KUKA KRL program: EPS_2_25862_MH04_A_20251016040658.src

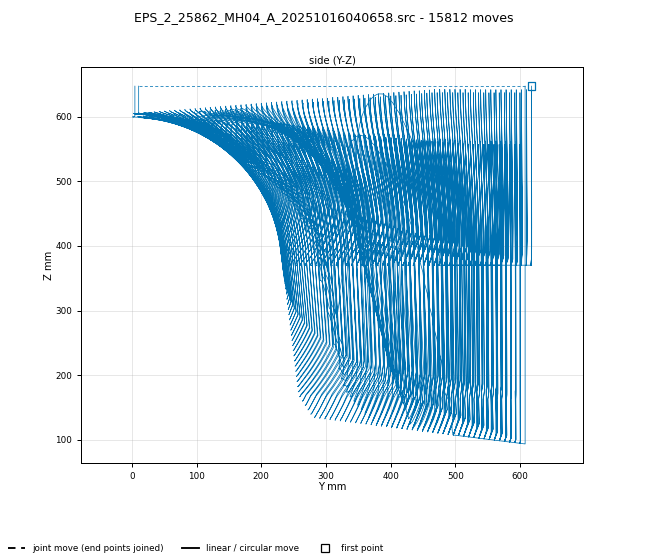
[picture p0: tool path of EPS_2_25862_MH04_A_20251016040658.src, 15812 of 15814 moves have a stored position in this frame; points joined in program order, loops and branches not executed]
&ACCESS RVP
&REL 4
&COMMENT QRS 19112012
&PARAM EDITMASK = *
DEF PART()
EXT BAS (BAS_COMMAND :IN,REAL :IN )
INT I
BAS (#INITMOV,0 )

;KUKA QRS Post kuka4.cps  Date:22-06-2017 !

File_ID=2885

QRS_PRE_INIT()

;Init var - Until changes are made in qrs_pre_init
Outlet_Square_prg=0
Inlet_1_Square_prg=0
Inlet_2_Square_prg=0
Inlet_3_Square_prg=0
Inlet_4_Square_prg=0
Inlet_5_Square_prg=0

Outlet_1={X 0.000, Y 466.000, Z 408.500, B 0.000, E1 0.000 }
Inlet_1={X 0.000, Y 522.780, Z 374.000, B 0.000, E1 180.000 }
Inlet_2={X 0.000, Y 522.780, Z 374.000, B 0.000, E1 270.000 }
Outlet_1_type=457
Inlet_1_type=366
Inlet_2_type=366
;QRS#1=Sidecore dimensions
;QRS#2=450-18" Concrete
;QRS#3=375-15" PVC SDR 35
;QRS#4=375-15" PVC SDR 35
;QRS#5=
;QRS#6=
;QRS#7=
;QRS#8=
;QRS#9=28A PSX-2
;QRS#10=20Y PSX
;QRS#11=20Y PSX
;QRS#12=
;QRS#13=
;QRS#14=
;QRS#15=
;QRS#16=1220x127x991 3,25'
;QRS#17=EPS Height
;QRS#18=637
;QRS#19=*
;QRS#20= UPDATED VERSION 22-06-2017
;QRS#21=*
Outlet_Square=0250
Inlet_1_Square=0250
Inlet_2_Square=0250
Inlet_3_Square=0
Inlet_4_Square=0
Inlet_5_Square=0
Mill_Square=1
Outlet_Square_Prg=274
Inlet_1_Square_prg=252
Inlet_2_Square_prg=252

QRS_INIT()

$ADVANCE=5

; T1
PTP {E1 171.055,E2 171.055}
PTP {X 0,Y 617.763,A -85,B 0,C 180,E1 171.055,E2 171.055,E3 0,E4 0,E5 0,E6 0}
QRS_SPEED_INIT()
LIN {X 0,Y 617.763,Z 647,A -85,B 0,C 180,E1 171.055,E2 171.055,E3 0,E4 0,E5 0,E6 0} C_VEL
LIN {X 0,Y 617.763,Z 372.16,A -85,B 0,C 180,E1 171.055,E2 171.055} C_VEL
LIN {X 0,Y 617.801,Z 370.16,A -85,B 0,C 180,E1 171.241,E2 171.241} C_VEL
LIN {X 0,Y 617.985,Z 370.16,A -85,B 0,C 180,E1 171.886,E2 171.886} C_VEL
LIN {X 0,Y 618.056,Z 370.16,A -85,B 0,C 180,E1 176.532,E2 176.532} C_VEL
LIN {X 0,Y 618.006,Z 370.16,A -85,B 0,C 180,E1 181.155,E2 181.155} C_VEL
LIN {X 0,Y 617.998,Z 370.16,A -85,B 0,C 180,E1 185.786,E2 185.786} C_VEL
LIN {X 0,Y 617.999,Z 370.16,A -85,B 0,C 180,E1 190.456,E2 190.456} C_VEL
LIN {X 0,Y 617.933,Z 370.16,A -85,B 0,C 180,E1 195.198,E2 195.198} C_VEL
LIN {X 0,Y 617.958,Z 370.16,A -85,B 0,C 180,E1 200.048,E2 200.048} C_VEL
LIN {X 0,Y 617.454,Z 370.16,A -85,B 0,C 180,E1 202.548,E2 202.548} C_VEL
LIN {X 0,Y 617.878,Z 370.16,A -85,B 0,C 180,E1 205.058,E2 205.058} C_VEL
LIN {X 0,Y 617.387,Z 370.16,A -85,B 0,C 180,E1 207.661,E2 207.661} C_VEL
LIN {X 0,Y 617.859,Z 370.16,A -85,B 0,C 180,E1 210.279,E2 210.279} C_VEL
LIN {X 0,Y 617.331,Z 370.16,A -85,B 0,C 180,E1 213.026,E2 213.026} C_VEL
LIN {X 0,Y 617.826,Z 370.16,A -85,B 0,C 180,E1 215.797,E2 215.797} C_VEL
LIN {X 0,Y 617.905,Z 370.16,A -85,B 0,C 180,E1 218.696,E2 218.696} C_VEL
LIN {X 0,Y 617.423,Z 370.16,A -85,B 0,C 180,E1 221.762,E2 221.762} C_VEL
LIN {X 0,Y 617.856,Z 370.16,A -85,B 0,C 180,E1 224.903,E2 224.903} C_VEL
LIN {X 0,Y 617.741,Z 370.16,A -85,B 0,C 180,E1 228.278,E2 228.278} C_VEL
LIN {X 0,Y 617.537,Z 370.16,A -85,B 0,C 180,E1 231.278,E2 231.278} C_VEL
LIN {X 0,Y 617.566,Z 370.16,A -85,B 0,C 180,E1 231.901,E2 231.901} C_VEL
LIN {X 0,Y 617.813,Z 370.16,A -85,B 0,C 180,E1 234.203,E2 234.203} C_VEL
LIN {X 0,Y 617.312,Z 370.16,A -85,B 0,C 180,E1 236.974,E2 236.974} C_VEL
LIN {X 0,Y 617.839,Z 370.16,A -85,B 0,C 180,E1 239.721,E2 239.721} C_VEL
LIN {X 0,Y 618.074,Z 370.16,A -85,B 0,C 180,E1 244.633,E2 244.633} C_VEL
LIN {X 0,Y 617.706,Z 370.16,A -85,B 0,C 180,E1 244.776,E2 244.776} C_VEL
LIN {X 0,Y 617.081,Z 370.236,A -85,B 0,C 180,E1 244.869,E2 244.869} C_VEL
LIN {X 0,Y 617.72,Z 382.151,A -85,B 0,C 180,E1 245.046,E2 245.046} C_VEL
LIN {X 0,Y 617.911,Z 419.432,A -85,B 0,C 180,E1 245.531,E2 245.531} C_VEL
LIN {X 0,Y 617.851,Z 429.801,A -85,B 0,C 180,E1 245.698,E2 245.698} C_VEL
LIN {X 0,Y 617.803,Z 439.075,A -85,B 0,C 180,E1 245.882,E2 245.882} C_VEL
LIN {X 0,Y 617.897,Z 451.685,A -85,B 0,C 180,E1 246.204,E2 246.204} C_VEL
LIN {X 0,Y 617.827,Z 462.897,A -85,B 0,C 180,E1 246.539,E2 246.539} C_VEL
LIN {X 0,Y 617.935,Z 474.971,A -85,B 0,C 180,E1 246.971,E2 246.971} C_VEL
LIN {X 0,Y 617.943,Z 485.368,A -85,B 0,C 180,E1 247.392,E2 247.392} C_VEL
LIN {X 0,Y 617.874,Z 495.678,A -85,B 0,C 180,E1 247.859,E2 247.859} C_VEL
LIN {X 0,Y 617.945,Z 506.347,A -85,B 0,C 180,E1 248.407,E2 248.407} C_VEL
LIN {X 0,Y 617.966,Z 517.222,A -85,B 0,C 180,E1 249.028,E2 249.028} C_VEL
LIN {X 0,Y 617.937,Z 527.03,A -85,B 0,C 180,E1 249.644,E2 249.644} C_VEL
LIN {X 0,Y 617.951,Z 536.534,A -85,B 0,C 180,E1 250.302,E2 250.302} C_VEL
LIN {X 0,Y 617.957,Z 545.725,A -85,B 0,C 180,E1 250.999,E2 250.999} C_VEL
LIN {X 0,Y 617.962,Z 554.652,A -85,B 0,C 180,E1 251.74,E2 251.74} C_VEL
LIN {X 0,Y 617.941,Z 563.035,A -85,B 0,C 180,E1 252.497,E2 252.497} C_VEL
LIN {X 0,Y 617.895,Z 570.428,A -85,B 0,C 180,E1 253.221,E2 253.221} C_VEL
LIN {X 0,Y 617.949,Z 578.128,A -85,B 0,C 180,E1 254.047,E2 254.047} C_VEL
LIN {X 0,Y 617.971,Z 584.666,A -85,B 0,C 180,E1 254.803,E2 254.803} C_VEL
LIN {X 0,Y 617.883,Z 591.779,A -85,B 0,C 180,E1 255.697,E2 255.697} C_VEL
LIN {X 0,Y 617.867,Z 598.243,A -85,B 0,C 180,E1 256.59,E2 256.59} C_VEL
LIN {X 0,Y 617.969,Z 604.103,A -85,B 0,C 180,E1 257.481,E2 257.481} C_VEL
LIN {X 0,Y 617.879,Z 609.465,A -85,B 0,C 180,E1 258.365,E2 258.365} C_VEL
LIN {X 0,Y 617.831,Z 615.768,A -85,B 0,C 180,E1 259.542,E2 259.542} C_VEL
LIN {X 0,Y 617.911,Z 619.334,A -85,B 0,C 180,E1 260.281,E2 260.281} C_VEL
LIN {X 0,Y 617.927,Z 624.37,A -85,B 0,C 180,E1 261.452,E2 261.452} C_VEL
LIN {X 0,Y 617.83,Z 627.758,A -85,B 0,C 180,E1 262.351,E2 262.351} C_VEL
LIN {X 0,Y 617.871,Z 630.79,A -85,B 0,C 180,E1 263.283,E2 263.283} C_VEL
LIN {X 0,Y 617.981,Z 633.385,A -85,B 0,C 180,E1 264.214,E2 264.214} C_VEL
LIN {X 0,Y 617.916,Z 634.618,A -85,B 0,C 180,E1 264.678,E2 264.678} C_VEL
LIN {X 0,Y 617.792,Z 636.669,A -85,B 0,C 180,E1 265.605,E2 265.605} C_VEL
LIN {X 0,Y 617.811,Z 638.259,A -85,B 0,C 180,E1 266.531,E2 266.531} C_VEL
LIN {X 0,Y 617.948,Z 639.966,A -85,B 0,C 180,E1 267.92,E2 267.92} C_VEL
LIN {X 0,Y 617.798,Z 640.661,A -85,B 0,C 180,E1 268.845,E2 268.845} C_VEL
LIN {X 0,Y 617.834,Z 640.908,A -85,B 0,C 180,E1 270.232,E2 270.232} C_VEL
LIN {X 0,Y 617.983,Z 640.61,A -85,B 0,C 180,E1 271.156,E2 271.156} C_VEL
LIN {X 0,Y 617.815,Z 639.475,A -85,B 0,C 180,E1 272.544,E2 272.544} C_VEL
LIN {X 0,Y 617.845,Z 638.248,A -85,B 0,C 180,E1 273.469,E2 273.469} C_VEL
LIN {X 0,Y 617.914,Z 637.45,A -85,B 0,C 180,E1 273.932,E2 273.932} C_VEL
LIN {X 0,Y 617.842,Z 634.634,A -85,B 0,C 180,E1 275.324,E2 275.324} C_VEL
LIN {X 0,Y 617.779,Z 632.188,A -85,B 0,C 180,E1 276.254,E2 276.254} C_VEL
LIN {X 0,Y 617.944,Z 627.726,A -85,B 0,C 180,E1 277.649,E2 277.649} C_VEL
LIN {X 0,Y 617.874,Z 623.347,A -85,B 0,C 180,E1 278.796,E2 278.796} C_VEL
LIN {X 0,Y 617.822,Z 619.616,A -85,B 0,C 180,E1 279.666,E2 279.666} C_VEL
LIN {X 0,Y 617.937,Z 614.253,A -85,B 0,C 180,E1 280.751,E2 280.751} C_VEL
LIN {X 0,Y 617.944,Z 609.445,A -85,B 0,C 180,E1 281.634,E2 281.634} C_VEL
LIN {X 0,Y 617.865,Z 602.193,A -85,B 0,C 180,E1 282.818,E2 282.818} C_VEL
LIN {X 0,Y 617.94,Z 596.131,A -85,B 0,C 180,E1 283.707,E2 283.707} C_VEL
LIN {X 0,Y 617.957,Z 589.464,A -85,B 0,C 180,E1 284.6,E2 284.6} C_VEL
LIN {X 0,Y 617.88,Z 581.509,A -85,B 0,C 180,E1 285.571,E2 285.571} C_VEL
LIN {X 0,Y 617.913,Z 574.458,A -85,B 0,C 180,E1 286.356,E2 286.356} C_VEL
LIN {X 0,Y 617.964,Z 566.289,A -85,B 0,C 180,E1 287.188,E2 287.188} C_VEL
LIN {X 0,Y 617.928,Z 559.146,A -85,B 0,C 180,E1 287.864,E2 287.864} C_VEL
LIN {X 0,Y 617.92,Z 550.267,A -85,B 0,C 180,E1 288.633,E2 288.633} C_VEL
LIN {X 0,Y 617.942,Z 541.357,A -85,B 0,C 180,E1 289.339,E2 289.339} C_VEL
LIN {X 0,Y 617.96,Z 532.851,A -85,B 0,C 180,E1 289.96,E2 289.96} C_VEL
LIN {X 0,Y 617.949,Z 523.456,A -85,B 0,C 180,E1 290.588,E2 290.588} C_VEL
LIN {X 0,Y 617.919,Z 513.262,A -85,B 0,C 180,E1 291.207,E2 291.207} C_VEL
LIN {X 0,Y 617.945,Z 503.396,A -85,B 0,C 180,E1 291.75,E2 291.75} C_VEL
LIN {X 0,Y 617.963,Z 492.338,A -85,B 0,C 180,E1 292.294,E2 292.294} C_VEL
LIN {X 0,Y 617.929,Z 481.553,A -85,B 0,C 180,E1 292.769,E2 292.769} C_VEL
LIN {X 0,Y 617.813,Z 471.413,A -85,B 0,C 180,E1 293.169,E2 293.169} C_VEL
LIN {X 0,Y 617.936,Z 458.266,A -85,B 0,C 180,E1 293.602,E2 293.602} C_VEL
LIN {X 0,Y 617.915,Z 446.913,A -85,B 0,C 180,E1 293.922,E2 293.922} C_VEL
LIN {X 0,Y 617.746,Z 436.06,A -85,B 0,C 180,E1 294.184,E2 294.184} C_VEL
LIN {X 0,Y 617.908,Z 424.188,A -85,B 0,C 180,E1 294.398,E2 294.398} C_VEL
LIN {X 0,Y 617.873,Z 406.799,A -85,B 0,C 180,E1 294.638,E2 294.638} C_VEL
LIN {X 0,Y 617.621,Z 379.189,A -85,B 0,C 180,E1 294.995,E2 294.995} C_VEL
LIN {X 0,Y 617.066,Z 370.16,A -85,B 0,C 180,E1 295.133,E2 295.133} C_VEL
LIN {X 0,Y 617.707,Z 370.16,A -85,B 0,C 180,E1 295.225,E2 295.225} C_VEL
LIN {X 0,Y 618.075,Z 370.16,A -85,B 0,C 180,E1 295.369,E2 295.369} C_VEL
LIN {X 0,Y 617.989,Z 370.16,A -85,B 0,C 180,E1 297.632,E2 297.632} C_VEL
LIN {X 0,Y 617.43,Z 370.16,A -85,B 0,C 180,E1 300.303,E2 300.303} C_VEL
LIN {X 0,Y 617.934,Z 370.16,A -85,B 0,C 180,E1 302.99,E2 302.99} C_VEL
LIN {X 0,Y 617.673,Z 370.16,A -85,B 0,C 180,E1 305.808,E2 305.808} C_VEL
LIN {X 0,Y 617.667,Z 370.16,A -85,B 0,C 180,E1 308.111,E2 308.111} C_VEL
LIN {X 0,Y 617.76,Z 370.16,A -85,B 0,C 180,E1 311.734,E2 311.734} C_VEL
LIN {X 0,Y 617.402,Z 370.16,A -85,B 0,C 180,E1 315.055,E2 315.055} C_VEL
LIN {X 0,Y 617.766,Z 370.16,A -85,B 0,C 180,E1 318.276,E2 318.276} C_VEL
LIN {X 0,Y 617.372,Z 370.16,A -85,B 0,C 180,E1 321.925,E2 321.925} C_VEL
LIN {X 0,Y 617.835,Z 370.16,A -85,B 0,C 180,E1 324.203,E2 324.203} C_VEL
LIN {X 0,Y 617.363,Z 370.16,A -85,B 0,C 180,E1 326.976,E2 326.976} C_VEL
LIN {X 0,Y 617.895,Z 370.16,A -85,B 0,C 180,E1 329.723,E2 329.723} C_VEL
LIN {X 0,Y 617.432,Z 370.16,A -85,B 0,C 180,E1 332.342,E2 332.342} C_VEL
LIN {X 0,Y 617.927,Z 370.16,A -85,B 0,C 180,E1 334.945,E2 334.945} C_VEL
LIN {X 0,Y 618.05,Z 370.16,A -85,B 0,C 180,E1 339.647,E2 339.647} C_VEL
LIN {X 0,Y 617.925,Z 370.16,A -85,B 0,C 180,E1 339.797,E2 339.797} C_VEL
LIN {X 0,Y 617.569,Z 370.202,A -85,B 0,C 180,E1 339.878,E2 339.878} C_VEL
LIN {X 0,Y 617.849,Z 384.179,A -85,B 0,C 180,E1 340.078,E2 340.078} C_VEL
LIN {X 0,Y 617.994,Z 396.248,A -85,B 0,C 180,E1 340.32,E2 340.32} C_VEL
LIN {X 0,Y 618.025,Z 406.56,A -85,B 0,C 180,E1 340.58,E2 340.58} C_VEL
LIN {X 0,Y 617.971,Z 415.883,A -85,B 0,C 180,E1 340.858,E2 340.858} C_VEL
LIN {X 0,Y 617.923,Z 423.433,A -85,B 0,C 180,E1 341.114,E2 341.114} C_VEL
LIN {X 0,Y 617.995,Z 433.283,A -85,B 0,C 180,E1 341.505,E2 341.505} C_VEL
LIN {X 0,Y 617.986,Z 442.714,A -85,B 0,C 180,E1 341.929,E2 341.929} C_VEL
LIN {X 0,Y 617.95,Z 450.65,A -85,B 0,C 180,E1 342.327,E2 342.327} C_VEL
LIN {X 0,Y 617.997,Z 459.127,A -85,B 0,C 180,E1 342.801,E2 342.801} C_VEL
LIN {X 0,Y 617.99,Z 467.334,A -85,B 0,C 180,E1 343.309,E2 343.309} C_VEL
LIN {X 0,Y 617.994,Z 476.018,A -85,B 0,C 180,E1 343.905,E2 343.905} C_VEL
LIN {X 0,Y 617.979,Z 483.981,A -85,B 0,C 180,E1 344.508,E2 344.508} C_VEL
LIN {X 0,Y 617.963,Z 491.14,A -85,B 0,C 180,E1 345.102,E2 345.102} C_VEL
LIN {X 0,Y 617.968,Z 497.738,A -85,B 0,C 180,E1 345.699,E2 345.699} C_VEL
LIN {X 0,Y 618.003,Z 505.227,A -85,B 0,C 180,E1 346.443,E2 346.443} C_VEL
LIN {X 0,Y 617.949,Z 512.018,A -85,B 0,C 180,E1 347.184,E2 347.184} C_VEL
LIN {X 0,Y 617.926,Z 519.37,A -85,B 0,C 180,E1 348.071,E2 348.071} C_VEL
LIN {X 0,Y 617.997,Z 525.839,A -85,B 0,C 180,E1 348.956,E2 348.956} C_VEL
LIN {X 0,Y 617.946,Z 531.027,A -85,B 0,C 180,E1 349.739,E2 349.739} C_VEL
LIN {X 0,Y 617.876,Z 535.713,A -85,B 0,C 180,E1 350.519,E2 350.519} C_VEL
LIN {X 0,Y 617.912,Z 539.315,A -85,B 0,C 180,E1 351.182,E2 351.182} C_VEL
LIN {X 0,Y 617.988,Z 543.836,A -85,B 0,C 180,E1 352.119,E2 352.119} C_VEL
LIN {X 0,Y 617.903,Z 546.855,A -85,B 0,C 180,E1 352.817,E2 352.817} C_VEL
LIN {X 0,Y 617.832,Z 550.397,A -85,B 0,C 180,E1 353.747,E2 353.747} C_VEL
LIN {X 0,Y 617.917,Z 553.348,A -85,B 0,C 180,E1 354.677,E2 354.677} C_VEL
LIN {X 0,Y 617.967,Z 555.788,A -85,B 0,C 180,E1 355.605,E2 355.605} C_VEL
LIN {X 0,Y 617.847,Z 557.776,A -85,B 0,C 180,E1 356.531,E2 356.531} C_VEL
LIN {X 0,Y 617.856,Z 559.249,A -85,B 0,C 180,E1 357.457,E2 357.457} C_VEL
LIN {X 0,Y 617.914,Z 559.779,A -85,B 0,C 180,E1 357.92,E2 357.92} C_VEL
LIN {X 0,Y 617.944,Z 560.559,A -85,B 0,C 180,E1 358.845,E2 358.845} C_VEL
LIN {X 0,Y 617.88,Z 560.798,A -85,B 0,C 180,E1 359.307,E2 359.307} C_VEL
LIN {X 0,Y 617.825,Z 560.9,A -85,B 0,C 180,E1 360.231,E2 360.231} C_VEL
LIN {X 0,Y 617.894,Z 560.509,A -85,B 0,C 180,E1 361.156,E2 361.156} C_VEL
LIN {X 0,Y 617.881,Z 559.137,A -85,B 0,C 180,E1 362.543,E2 362.543} C_VEL
LIN {X 0,Y 617.822,Z 557.63,A -85,B 0,C 180,E1 363.469,E2 363.469} C_VEL
LIN {X 0,Y 617.899,Z 555.598,A -85,B 0,C 180,E1 364.395,E2 364.395} C_VEL
LIN {X 0,Y 617.955,Z 553.067,A -85,B 0,C 180,E1 365.322,E2 365.322} C_VEL
LIN {X 0,Y 617.87,Z 550.053,A -85,B 0,C 180,E1 366.252,E2 366.252} C_VEL
LIN {X 0,Y 617.941,Z 545.458,A -85,B 0,C 180,E1 367.415,E2 367.415} C_VEL
LIN {X 0,Y 617.978,Z 542.3,A -85,B 0,C 180,E1 368.115,E2 368.115} C_VEL
LIN {X 0,Y 617.885,Z 537.344,A -85,B 0,C 180,E1 369.091,E2 369.091} C_VEL
LIN {X 0,Y 617.884,Z 534.05,A -85,B 0,C 180,E1 369.676,E2 369.676} C_VEL
LIN {X 0,Y 617.956,Z 529.189,A -85,B 0,C 180,E1 370.457,E2 370.457} C_VEL
LIN {X 0,Y 617.992,Z 524.162,A -85,B 0,C 180,E1 371.191,E2 371.191} C_VEL
LIN {X 0,Y 617.927,Z 518.64,A -85,B 0,C 180,E1 371.929,E2 371.929} C_VEL
LIN {X 0,Y 617.936,Z 512.535,A -85,B 0,C 180,E1 372.668,E2 372.668} C_VEL
LIN {X 0,Y 617.996,Z 505.794,A -85,B 0,C 180,E1 373.408,E2 373.408} C_VEL
LIN {X 0,Y 617.987,Z 499.923,A -85,B 0,C 180,E1 374.003,E2 374.003} C_VEL
LIN {X 0,Y 617.964,Z 493.532,A -85,B 0,C 180,E1 374.6,E2 374.6} C_VEL
LIN {X 0,Y 617.969,Z 486.545,A -85,B 0,C 180,E1 375.197,E2 375.197} C_VEL
LIN {X 0,Y 617.969,Z 478.994,A -85,B 0,C 180,E1 375.788,E2 375.788} C_VEL
LIN {X 0,Y 618.002,Z 470.17,A -85,B 0,C 180,E1 376.412,E2 376.412} C_VEL
LIN {X 0,Y 617.987,Z 463.836,A -85,B 0,C 180,E1 376.824,E2 376.824} C_VEL
LIN {X 0,Y 617.993,Z 454.31,A -85,B 0,C 180,E1 377.382,E2 377.382} C_VEL
LIN {X 0,Y 617.954,Z 446.299,A -85,B 0,C 180,E1 377.806,E2 377.806} C_VEL
LIN {X 0,Y 618.005,Z 437.901,A -85,B 0,C 180,E1 378.203,E2 378.203} C_VEL
LIN {X 0,Y 617.997,Z 428.224,A -85,B 0,C 180,E1 378.609,E2 378.609} C_VEL
LIN {X 0,Y 617.916,Z 419.62,A -85,B 0,C 180,E1 378.929,E2 378.929} C_VEL
LIN {X 0,Y 617.991,Z 410.198,A -85,B 0,C 180,E1 379.228,E2 379.228} C_VEL
LIN {X 0,Y 617.991,Z 400.635,A -85,B 0,C 180,E1 379.486,E2 379.486} C_VEL
LIN {X 0,Y 617.933,Z 390.91,A -85,B 0,C 180,E1 379.704,E2 379.704} C_VEL
LIN {X 0,Y 617.689,Z 380.946,A -85,B 0,C 180,E1 379.884,E2 379.884} C_VEL
LIN {X 0,Y 617.047,Z 370.16,A -85,B 0,C 180,E1 380.058,E2 380.058} C_VEL
LIN {X 0,Y 618.002,Z 370.16,A -85,B 0,C 180,E1 380.355,E2 380.355} C_VEL
LIN {X 0,Y 617.929,Z 370.16,A -85,B 0,C 180,E1 385.055,E2 385.055} C_VEL
LIN {X 0,Y 617.437,Z 370.16,A -85,B 0,C 180,E1 387.658,E2 387.658} C_VEL
LIN {X 0,Y 617.899,Z 370.16,A -85,B 0,C 180,E1 390.277,E2 390.277} C_VEL
LIN {X 0,Y 617.367,Z 370.16,A -85,B 0,C 180,E1 393.024,E2 393.024} C_VEL
LIN {X 0,Y 617.838,Z 370.16,A -85,B 0,C 180,E1 395.797,E2 395.797} C_VEL
LIN {X 0,Y 617.935,Z 370.16,A -85,B 0,C 180,E1 398.693,E2 398.693} C_VEL
LIN {X 0,Y 617.441,Z 370.16,A -85,B 0,C 180,E1 401.76,E2 401.76} C_VEL
LIN {X 0,Y 617.851,Z 370.16,A -85,B 0,C 180,E1 404.903,E2 404.903} C_VEL
LIN {X 0,Y 617.765,Z 370.16,A -85,B 0,C 180,E1 408.275,E2 408.275} C_VEL
LIN {X 0,Y 617.553,Z 370.16,A -85,B 0,C 180,E1 411.278,E2 411.278} C_VEL
LIN {X 0,Y 617.579,Z 370.16,A -85,B 0,C 180,E1 411.9,E2 411.9} C_VEL
LIN {X 0,Y 617.823,Z 370.16,A -85,B 0,C 180,E1 414.202,E2 414.202} C_VEL
LIN {X 0,Y 617.352,Z 370.16,A -85,B 0,C 180,E1 416.975,E2 416.975} C_VEL
LIN {X 0,Y 617.884,Z 370.16,A -85,B 0,C 180,E1 419.722,E2 419.722} C_VEL
LIN {X 0,Y 617.423,Z 370.16,A -85,B 0,C 180,E1 422.341,E2 422.341} C_VEL
LIN {X 0,Y 617.919,Z 370.16,A -85,B 0,C 180,E1 424.944,E2 424.944} C_VEL
LIN {X 0,Y 618.043,Z 370.16,A -85,B 0,C 180,E1 429.646,E2 429.646} C_VEL
LIN {X 0,Y 617.917,Z 370.16,A -85,B 0,C 180,E1 429.796,E2 429.796} C_VEL
LIN {X 0,Y 617.553,Z 370.168,A -85,B 0,C 180,E1 429.877,E2 429.877} C_VEL
LIN {X 0,Y 617.839,Z 384.153,A -85,B 0,C 180,E1 430.077,E2 430.077} C_VEL
LIN {X 0,Y 617.985,Z 395.303,A -85,B 0,C 180,E1 430.298,E2 430.298} C_VEL
LIN {X 0,Y 618.023,Z 406.525,A -85,B 0,C 180,E1 430.579,E2 430.579} C_VEL
LIN {X 0,Y 617.975,Z 415.849,A -85,B 0,C 180,E1 430.857,E2 430.857} C_VEL
LIN {X 0,Y 617.927,Z 423.396,A -85,B 0,C 180,E1 431.113,E2 431.113} C_VEL
LIN {X 0,Y 618.007,Z 433.84,A -85,B 0,C 180,E1 431.53,E2 431.53} C_VEL
LIN {X 0,Y 617.989,Z 442.695,A -85,B 0,C 180,E1 431.929,E2 431.929} C_VEL
LIN {X 0,Y 617.954,Z 450.641,A -85,B 0,C 180,E1 432.326,E2 432.326} C_VEL
LIN {X 0,Y 618,Z 459.118,A -85,B 0,C 180,E1 432.801,E2 432.801} C_VEL
LIN {X 0,Y 617.992,Z 467.324,A -85,B 0,C 180,E1 433.308,E2 433.308} C_VEL
LIN {X 0,Y 617.996,Z 476.144,A -85,B 0,C 180,E1 433.914,E2 433.914} C_VEL
LIN {X 0,Y 617.979,Z 483.974,A -85,B 0,C 180,E1 434.507,E2 434.507} C_VEL
LIN {X 0,Y 617.962,Z 491.135,A -85,B 0,C 180,E1 435.101,E2 435.101} C_VEL
LIN {X 0,Y 617.967,Z 497.734,A -85,B 0,C 180,E1 435.698,E2 435.698} C_VEL
LIN {X 0,Y 618.001,Z 505.223,A -85,B 0,C 180,E1 436.443,E2 436.443} C_VEL
LIN {X 0,Y 617.948,Z 512.014,A -85,B 0,C 180,E1 437.183,E2 437.183} C_VEL
LIN {X 0,Y 617.925,Z 519.367,A -85,B 0,C 180,E1 438.07,E2 438.07} C_VEL
LIN {X 0,Y 617.996,Z 525.836,A -85,B 0,C 180,E1 438.956,E2 438.956} C_VEL
LIN {X 0,Y 617.946,Z 531.023,A -85,B 0,C 180,E1 439.738,E2 439.738} C_VEL
LIN {X 0,Y 617.878,Z 535.707,A -85,B 0,C 180,E1 440.518,E2 440.518} C_VEL
LIN {X 0,Y 617.932,Z 540.659,A -85,B 0,C 180,E1 441.455,E2 441.455} C_VEL
LIN {X 0,Y 617.961,Z 544.837,A -85,B 0,C 180,E1 442.351,E2 442.351} C_VEL
LIN {X 0,Y 617.904,Z 546.853,A -85,B 0,C 180,E1 442.817,E2 442.817} C_VEL
LIN {X 0,Y 617.83,Z 550.395,A -85,B 0,C 180,E1 443.747,E2 443.747} C_VEL
LIN {X 0,Y 617.912,Z 553.348,A -85,B 0,C 180,E1 444.677,E2 444.677} C_VEL
LIN {X 0,Y 617.959,Z 555.789,A -85,B 0,C 180,E1 445.605,E2 445.605} C_VEL
LIN {X 0,Y 617.84,Z 557.777,A -85,B 0,C 180,E1 446.531,E2 446.531} C_VEL
LIN {X 0,Y 617.849,Z 559.25,A -85,B 0,C 180,E1 447.456,E2 447.456} C_VEL
LIN {X 0,Y 617.94,Z 560.56,A -85,B 0,C 180,E1 448.844,E2 448.844} C_VEL
LIN {X 0,Y 617.843,Z 560.918,A -85,B 0,C 180,E1 449.768,E2 449.768} C_VEL
LIN {X 0,Y 617.863,Z 560.782,A -85,B 0,C 180,E1 450.693,E2 450.693} C_VEL
LIN {X 0,Y 617.911,Z 560.504,A -85,B 0,C 180,E1 451.155,E2 451.155} C_VEL
LIN {X 0,Y 617.956,Z 559.662,A -85,B 0,C 180,E1 452.08,E2 452.08} C_VEL
LIN {X 0,Y 617.903,Z 559.132,A -85,B 0,C 180,E1 452.542,E2 452.542} C_VEL
LIN {X 0,Y 617.845,Z 557.625,A -85,B 0,C 180,E1 453.468,E2 453.468} C_VEL
LIN {X 0,Y 617.922,Z 555.594,A -85,B 0,C 180,E1 454.394,E2 454.394} C_VEL
LIN {X 0,Y 617.976,Z 553.064,A -85,B 0,C 180,E1 455.322,E2 455.322} C_VEL
LIN {X 0,Y 617.884,Z 550.052,A -85,B 0,C 180,E1 456.252,E2 456.252} C_VEL
LIN {X 0,Y 617.946,Z 545.459,A -85,B 0,C 180,E1 457.415,E2 457.415} C_VEL
LIN {X 0,Y 617.981,Z 542.302,A -85,B 0,C 180,E1 458.114,E2 458.114} C_VEL
LIN {X 0,Y 617.886,Z 537.337,A -85,B 0,C 180,E1 459.092,E2 459.092} C_VEL
LIN {X 0,Y 617.886,Z 534.047,A -85,B 0,C 180,E1 459.676,E2 459.676} C_VEL
LIN {X 0,Y 617.957,Z 529.193,A -85,B 0,C 180,E1 460.456,E2 460.456} C_VEL
LIN {X 0,Y 617.992,Z 524.167,A -85,B 0,C 180,E1 461.19,E2 461.19} C_VEL
LIN {X 0,Y 617.927,Z 518.646,A -85,B 0,C 180,E1 461.929,E2 461.929} C_VEL
LIN {X 0,Y 617.936,Z 512.542,A -85,B 0,C 180,E1 462.668,E2 462.668} C_VEL
LIN {X 0,Y 617.996,Z 505.8,A -85,B 0,C 180,E1 463.408,E2 463.408} C_VEL
LIN {X 0,Y 617.987,Z 499.93,A -85,B 0,C 180,E1 464.002,E2 464.002} C_VEL
LIN {X 0,Y 617.964,Z 493.54,A -85,B 0,C 180,E1 464.599,E2 464.599} C_VEL
LIN {X 0,Y 617.968,Z 486.554,A -85,B 0,C 180,E1 465.197,E2 465.197} C_VEL
LIN {X 0,Y 617.969,Z 478.992,A -85,B 0,C 180,E1 465.788,E2 465.788} C_VEL
LIN {X 0,Y 618.004,Z 470.529,A -85,B 0,C 180,E1 466.388,E2 466.388} C_VEL
LIN {X 0,Y 617.994,Z 462.677,A -85,B 0,C 180,E1 466.894,E2 466.894} C_VEL
LIN {X 0,Y 617.99,Z 455.815,A -85,B 0,C 180,E1 467.3,E2 467.3} C_VEL
LIN {X 0,Y 617.942,Z 447.397,A -85,B 0,C 180,E1 467.753,E2 467.753} C_VEL
LIN {X 0,Y 618.002,Z 438.211,A -85,B 0,C 180,E1 468.19,E2 468.19} C_VEL
LIN {X 0,Y 617.997,Z 428.217,A -85,B 0,C 180,E1 468.61,E2 468.61} C_VEL
LIN {X 0,Y 617.906,Z 419.095,A -85,B 0,C 180,E1 468.947,E2 468.947} C_VEL
LIN {X 0,Y 618.003,Z 409.603,A -85,B 0,C 180,E1 469.244,E2 469.244} C_VEL
LIN {X 0,Y 618.009,Z 400.729,A -85,B 0,C 180,E1 469.483,E2 469.483} C_VEL
LIN {X 0,Y 617.951,Z 391.726,A -85,B 0,C 180,E1 469.687,E2 469.687} C_VEL
LIN {X 0,Y 617.738,Z 381.514,A -85,B 0,C 180,E1 469.875,E2 469.875} C_VEL
LIN {X 0,Y 617.07,Z 370.16,A -85,B 0,C 180,E1 470.055,E2 470.055} C_VEL
LIN {X 0,Y 617.214,Z 370.16,A -85,B 0,C 180,E1 470.073,E2 470.073} C_VEL
LIN {X 0,Y 617.999,Z 370.16,A -85,B 0,C 180,E1 472.526,E2 472.526} C_VEL
LIN {X 0,Y 617.417,Z 370.16,A -85,B 0,C 180,E1 475.077,E2 475.077} C_VEL
LIN {X 0,Y 617.839,Z 370.16,A -85,B 0,C 180,E1 477.638,E2 477.638} C_VEL
LIN {X 0,Y 617.328,Z 370.16,A -85,B 0,C 180,E1 480.307,E2 480.307} C_VEL
LIN {X 0,Y 617.804,Z 370.16,A -85,B 0,C 180,E1 482.996,E2 482.996} C_VEL
LIN {X 0,Y 617.664,Z 370.16,A -85,B 0,C 180,E1 484.19,E2 484.19} C_VEL
LIN {X 0,Y 617.749,Z 370.16,A -85,B 0,C 180,E1 488.706,E2 488.706} C_VEL
LIN {X 0,Y 617.414,Z 370.16,A -85,B 0,C 180,E1 491.761,E2 491.761} C_VEL
LIN {X 0,Y 617.835,Z 370.16,A -85,B 0,C 180,E1 494.903,E2 494.903} C_VEL
LIN {X 0,Y 617.756,Z 370.16,A -85,B 0,C 180,E1 498.275,E2 498.275} C_VEL
LIN {X 0,Y 617.524,Z 370.16,A -85,B 0,C 180,E1 501.276,E2 501.276} C_VEL
LIN {X 0,Y 617.765,Z 370.16,A -85,B 0,C 180,E1 504.198,E2 504.198} C_VEL
LIN {X 0,Y 617.288,Z 370.16,A -85,B 0,C 180,E1 506.971,E2 506.971} C_VEL
LIN {X 0,Y 617.835,Z 370.16,A -85,B 0,C 180,E1 509.719,E2 509.719} C_VEL
LIN {X 0,Y 617.406,Z 370.16,A -85,B 0,C 180,E1 512.34,E2 512.34} C_VEL
LIN {X 0,Y 617.928,Z 370.16,A -85,B 0,C 180,E1 514.945,E2 514.945} C_VEL
LIN {X 0,Y 617.445,Z 370.16,A -85,B 0,C 180,E1 517.452,E2 517.452} C_VEL
LIN {X 0,Y 617.92,Z 370.16,A -85,B 0,C 180,E1 519.95,E2 519.95} C_VEL
LIN {X 0,Y 617.688,Z 370.16,A -85,B 0,C 180,E1 522.385,E2 522.385} C_VEL
LIN {X 0,Y 617.777,Z 370.16,A -85,B 0,C 180,E1 524.798,E2 524.798} C_VEL
LIN {X 0,Y 617.951,Z 370.16,A -85,B 0,C 180,E1 527.184,E2 527.184} C_VEL
LIN {X 0,Y 617.801,Z 370.16,A -85,B 0,C 180,E1 531.241,E2 531.241} C_VEL
LIN {X 0,Y 615.29,Z 370.16,A -85,B 0,C 180,E1 532.437,E2 532.437} C_VEL
LIN {X 0,Y 609.718,Z 370.16,A -85,B 0,C 180,E1 534.226,E2 534.226} C_VEL
LIN {X 0,Y 609.633,Z 370.16,A -85,B 0,C 180,E1 534.433,E2 534.433} C_VEL
LIN {X 0,Y 609.638,Z 370.16,A -85,B 0,C 180,E1 538.578,E2 538.578} C_VEL
LIN {X 0,Y 609.647,Z 370.16,A -85,B 0,C 180,E1 542.848,E2 542.848} C_VEL
LIN {X 0,Y 609.696,Z 370.16,A -85,B 0,C 180,E1 547.133,E2 547.133} C_VEL
LIN {X 0,Y 609.757,Z 370.16,A -85,B 0,C 180,E1 551.457,E2 551.457} C_VEL
LIN {X 0,Y 609.776,Z 370.16,A -85,B 0,C 180,E1 555.85,E2 555.85} C_VEL
LIN {X 0,Y 609.961,Z 370.16,A -85,B 0,C 180,E1 560.334,E2 560.334} C_VEL
LIN {X 0,Y 609.964,Z 370.16,A -85,B 0,C 180,E1 564.958,E2 564.958} C_VEL
LIN {X 0,Y 609.779,Z 370.16,A -85,B 0,C 180,E1 569.773,E2 569.773} C_VEL
LIN {X 0,Y 609.822,Z 370.16,A -85,B 0,C 180,E1 576.571,E2 576.571} C_VEL
LIN {X 0,Y 609.534,Z 370.16,A -85,B 0,C 180,E1 581.827,E2 581.827} C_VEL
LIN {X 0,Y 609.69,Z 370.16,A -85,B 0,C 180,E1 586.063,E2 586.063} C_VEL
LIN {X 0,Y 609.661,Z 370.16,A -85,B 0,C 180,E1 591.622,E2 591.622} C_VEL
LIN {X 0,Y 609.405,Z 370.16,A -85,B 0,C 180,E1 596.868,E2 596.868} C_VEL
LIN {X 0,Y 609.73,Z 370.16,A -85,B 0,C 180,E1 600.347,E2 600.347} C_VEL
LIN {X 0,Y 610.021,Z 370.16,A -85,B 0,C 180,E1 604.539,E2 604.539} C_VEL
LIN {X 0,Y 610.563,Z 440.168,A -85,B 0,C 180,E1 605.605,E2 605.605} C_VEL
LIN {X 0,Y 610.591,Z 476.06,A -85,B 0,C 180,E1 606.722,E2 606.722} C_VEL
LIN {X 0,Y 610.479,Z 510.256,A -85,B 0,C 180,E1 608.351,E2 608.351} C_VEL
LIN {X 0,Y 610.358,Z 543.138,A -85,B 0,C 180,E1 610.544,E2 610.544} C_VEL
LIN {X 0,Y 610.182,Z 572.739,A -85,B 0,C 180,E1 613.234,E2 613.234} C_VEL
LIN {X 0,Y 610.083,Z 596.969,A -85,B 0,C 180,E1 616.179,E2 616.179} C_VEL
LIN {X 0,Y 610.021,Z 615.714,A -85,B 0,C 180,E1 619.271,E2 619.271} C_VEL
LIN {X 0,Y 610.017,Z 629.454,A -85,B 0,C 180,E1 622.511,E2 622.511} C_VEL
LIN {X 0,Y 609.974,Z 637.968,A -85,B 0,C 180,E1 625.728,E2 625.728} C_VEL
LIN {X 0,Y 610.021,Z 641.505,A -85,B 0,C 180,E1 628.576,E2 628.576} C_VEL
LIN {X 0,Y 610.116,Z 641.508,A -85,B 0,C 180,E1 631.42,E2 631.42} C_VEL
LIN {X 0,Y 610.006,Z 636.457,A -85,B 0,C 180,E1 634.981,E2 634.981} C_VEL
LIN {X 0,Y 610.079,Z 625.508,A -85,B 0,C 180,E1 638.561,E2 638.561} C_VEL
LIN {X 0,Y 610.104,Z 608.729,A -85,B 0,C 180,E1 641.992,E2 641.992} C_VEL
LIN {X 0,Y 610.172,Z 587.268,A -85,B 0,C 180,E1 645.102,E2 645.102} C_VEL
LIN {X 0,Y 610.249,Z 560.619,A -85,B 0,C 180,E1 647.97,E2 647.97} C_VEL
LIN {X 0,Y 610.393,Z 530.052,A -85,B 0,C 180,E1 650.411,E2 650.411} C_VEL
LIN {X 0,Y 610.536,Z 497.801,A -85,B 0,C 180,E1 652.313,E2 652.313} C_VEL
LIN {X 0,Y 610.658,Z 461.459,A -85,B 0,C 180,E1 653.803,E2 653.803} C_VEL
LIN {X 0,Y 610.722,Z 425.817,A -85,B 0,C 180,E1 654.68,E2 654.68} C_VEL
LIN {X 0,Y 610.145,Z 370.16,A -85,B 0,C 180,E1 655.491,E2 655.491} C_VEL
LIN {X 0,Y 609.556,Z 370.16,A -85,B 0,C 180,E1 659.782,E2 659.782} C_VEL
LIN {X 0,Y 610.011,Z 370.16,A -85,B 0,C 180,E1 663.09,E2 663.09} C_VEL
LIN {X 0,Y 609.699,Z 370.16,A -85,B 0,C 180,E1 668.37,E2 668.37} C_VEL
LIN {X 0,Y 609.717,Z 370.16,A -85,B 0,C 180,E1 672.096,E2 672.096} C_VEL
LIN {X 0,Y 609.806,Z 370.16,A -85,B 0,C 180,E1 678.138,E2 678.138} C_VEL
LIN {X 0,Y 609.665,Z 370.16,A -85,B 0,C 180,E1 683.418,E2 683.418} C_VEL
LIN {X 0,Y 609.624,Z 370.16,A -85,B 0,C 180,E1 688.566,E2 688.566} C_VEL
LIN {X 0,Y 609.607,Z 370.16,A -85,B 0,C 180,E1 693.447,E2 693.447} C_VEL
LIN {X 0,Y 609.582,Z 370.16,A -85,B 0,C 180,E1 696.763,E2 696.763} C_VEL
LIN {X 0,Y 610.135,Z 370.331,A -85,B 0,C 180,E1 699.625,E2 699.625} C_VEL
LIN {X 0,Y 610.558,Z 406.298,A -85,B 0,C 180,E1 700.325,E2 700.325} C_VEL
LIN {X 0,Y 610.44,Z 438.962,A -85,B 0,C 180,E1 701.519,E2 701.519} C_VEL
LIN {X 0,Y 610.354,Z 469.557,A -85,B 0,C 180,E1 703.24,E2 703.24} C_VEL
LIN {X 0,Y 610.244,Z 496.282,A -85,B 0,C 180,E1 705.352,E2 705.352} C_VEL
LIN {X 0,Y 610.137,Z 520.488,A -85,B 0,C 180,E1 708.005,E2 708.005} C_VEL
LIN {X 0,Y 610.069,Z 538.091,A -85,B 0,C 180,E1 710.717,E2 710.717} C_VEL
LIN {X 0,Y 610.024,Z 550.94,A -85,B 0,C 180,E1 713.586,E2 713.586} C_VEL
LIN {X 0,Y 610.042,Z 558.69,A -85,B 0,C 180,E1 716.442,E2 716.442} C_VEL
LIN {X 0,Y 610.098,Z 561.447,A -85,B 0,C 180,E1 718.577,E2 718.577} C_VEL
LIN {X 0,Y 610.047,Z 561.385,A -85,B 0,C 180,E1 721.421,E2 721.421} C_VEL
LIN {X 0,Y 610.05,Z 556.976,A -85,B 0,C 180,E1 724.269,E2 724.269} C_VEL
LIN {X 0,Y 610.147,Z 546.376,A -85,B 0,C 180,E1 727.484,E2 727.484} C_VEL
LIN {X 0,Y 610.176,Z 530.078,A -85,B 0,C 180,E1 730.542,E2 730.542} C_VEL
LIN {X 0,Y 610.229,Z 509.076,A -85,B 0,C 180,E1 733.266,E2 733.266} C_VEL
LIN {X 0,Y 610.289,Z 483.558,A -85,B 0,C 180,E1 735.648,E2 735.648} C_VEL
LIN {X 0,Y 610.39,Z 454.566,A -85,B 0,C 180,E1 737.593,E2 737.593} C_VEL
LIN {X 0,Y 610.435,Z 421.781,A -85,B 0,C 180,E1 739.098,E2 739.098} C_VEL
LIN {X 0,Y 610.431,Z 387.592,A -85,B 0,C 180,E1 740.021,E2 740.021} C_VEL
LIN {X 0,Y 609.735,Z 370.16,A -85,B 0,C 180,E1 740.34,E2 740.34} C_VEL
LIN {X 0,Y 609.997,Z 370.16,A -85,B 0,C 180,E1 744.954,E2 744.954} C_VEL
LIN {X 0,Y 609.818,Z 370.16,A -85,B 0,C 180,E1 749.768,E2 749.768} C_VEL
LIN {X 0,Y 609.81,Z 370.16,A -85,B 0,C 180,E1 756.57,E2 756.57} C_VEL
LIN {X 0,Y 609.591,Z 370.16,A -85,B 0,C 180,E1 760.217,E2 760.217} C_VEL
LIN {X 0,Y 609.697,Z 370.16,A -85,B 0,C 180,E1 766.06,E2 766.06} C_VEL
LIN {X 0,Y 609.538,Z 370.16,A -85,B 0,C 180,E1 770.347,E2 770.347} C_VEL
LIN {X 0,Y 609.612,Z 370.16,A -85,B 0,C 180,E1 775.169,E2 775.169} C_VEL
LIN {X 0,Y 609.788,Z 370.16,A -85,B 0,C 180,E1 780.333,E2 780.333} C_VEL
LIN {X 0,Y 609.988,Z 370.16,A -85,B 0,C 180,E1 785.046,E2 785.046} C_VEL
LIN {X 0,Y 610.15,Z 370.569,A -85,B 0,C 180,E1 789.628,E2 789.628} C_VEL
LIN {X 0,Y 610.565,Z 407.218,A -85,B 0,C 180,E1 790.352,E2 790.352} C_VEL
LIN {X 0,Y 610.471,Z 440.068,A -85,B 0,C 180,E1 791.569,E2 791.569} C_VEL
LIN {X 0,Y 610.334,Z 470.978,A -85,B 0,C 180,E1 793.335,E2 793.335} C_VEL
LIN {X 0,Y 610.24,Z 498.045,A -85,B 0,C 180,E1 795.521,E2 795.521} C_VEL
LIN {X 0,Y 610.16,Z 521.847,A -85,B 0,C 180,E1 798.19,E2 798.19} C_VEL
LIN {X 0,Y 610.109,Z 540.064,A -85,B 0,C 180,E1 801.08,E2 801.08} C_VEL
LIN {X 0,Y 610.036,Z 552.167,A -85,B 0,C 180,E1 803.947,E2 803.947} C_VEL
LIN {X 0,Y 610.007,Z 559.886,A -85,B 0,C 180,E1 807.157,E2 807.157} C_VEL
LIN {X 0,Y 610.015,Z 561.996,A -85,B 0,C 180,E1 810.002,E2 810.002} C_VEL
LIN {X 0,Y 610.042,Z 559.728,A -85,B 0,C 180,E1 812.847,E2 812.847} C_VEL
LIN {X 0,Y 610.09,Z 551.752,A -85,B 0,C 180,E1 816.092,E2 816.092} C_VEL
LIN {X 0,Y 610.089,Z 539.551,A -85,B 0,C 180,E1 818.924,E2 818.924} C_VEL
LIN {X 0,Y 610.164,Z 521.154,A -85,B 0,C 180,E1 821.814,E2 821.814} C_VEL
LIN {X 0,Y 610.249,Z 498.276,A -85,B 0,C 180,E1 824.366,E2 824.366} C_VEL
LIN {X 0,Y 610.36,Z 470.953,A -85,B 0,C 180,E1 826.576,E2 826.576} C_VEL
LIN {X 0,Y 610.448,Z 440.048,A -85,B 0,C 180,E1 828.342,E2 828.342} C_VEL
LIN {X 0,Y 610.556,Z 408.022,A -85,B 0,C 180,E1 829.535,E2 829.535} C_VEL
LIN {X 0,Y 609.78,Z 372.806,A -85,B 0,C 180,E1 830.267,E2 830.267} C_VEL
LIN {X 0,Y 609.366,Z 370.16,A -85,B 0,C 180,E1 830.356,E2 830.356} C_VEL
LIN {X 0,Y 609.757,Z 370.16,A -85,B 0,C 180,E1 833.409,E2 833.409} C_VEL
LIN {X 0,Y 609.743,Z 370.16,A -85,B 0,C 180,E1 838.15,E2 838.15} C_VEL
LIN {X 0,Y 609.88,Z 370.16,A -85,B 0,C 180,E1 843.103,E2 843.103} C_VEL
LIN {X 0,Y 609.573,Z 370.16,A -85,B 0,C 180,E1 849.656,E2 849.656} C_VEL
LIN {X 0,Y 609.695,Z 370.16,A -85,B 0,C 180,E1 855.954,E2 855.954} C_VEL
LIN {X 0,Y 609.516,Z 370.16,A -85,B 0,C 180,E1 860.356,E2 860.356} C_VEL
LIN {X 0,Y 609.55,Z 370.16,A -85,B 0,C 180,E1 865.165,E2 865.165} C_VEL
LIN {X 0,Y 609.723,Z 370.16,A -85,B 0,C 180,E1 870.352,E2 870.352} C_VEL
LIN {X 0,Y 610.008,Z 370.16,A -85,B 0,C 180,E1 875.046,E2 875.046} C_VEL
LIN {X 0,Y 609.794,Z 370.16,A -85,B 0,C 180,E1 881.172,E2 881.172} C_VEL
LIN {X 0,Y 610.04,Z 370.16,A -85,B 0,C 180,E1 887.095,E2 887.095} C_VEL
LIN {X 0,Y 609.773,Z 370.16,A -85,B 0,C 180,E1 892.87,E2 892.87} C_VEL
LIN {X 0,Y 609.633,Z 370.16,A -85,B 0,C 180,E1 894.433,E2 894.433} C_VEL
LIN {X 0,Y 605.878,Z 370.16,A -85,B 0,C 180,E1 896.04,E2 896.04} C_VEL
LIN {X 0,Y 601.868,Z 370.16,A -85,B 0,C 180,E1 897.667,E2 897.667} C_VEL
LIN {X 0,Y 602.103,Z 370.16,A -85,B 0,C 180,E1 901.442,E2 901.442} C_VEL
LIN {X 0,Y 602.15,Z 370.16,A -85,B 0,C 180,E1 905.773,E2 905.773} C_VEL
LIN {X 0,Y 601.828,Z 370.16,A -85,B 0,C 180,E1 911.611,E2 911.611} C_VEL
LIN {X 0,Y 601.811,Z 370.16,A -85,B 0,C 180,E1 916.065,E2 916.065} C_VEL
LIN {X 0,Y 601.746,Z 370.16,A -85,B 0,C 180,E1 921.422,E2 921.422} C_VEL
LIN {X 0,Y 601.942,Z 370.16,A -85,B 0,C 180,E1 925.314,E2 925.314} C_VEL
LIN {X 0,Y 601.691,Z 370.16,A -85,B 0,C 180,E1 931.183,E2 931.183} C_VEL
LIN {X 0,Y 601.88,Z 370.16,A -85,B 0,C 180,E1 937.134,E2 937.134} C_VEL
LIN {X 0,Y 601.61,Z 370.16,A -85,B 0,C 180,E1 943.129,E2 943.129} C_VEL
LIN {X 0,Y 601.753,Z 370.16,A -85,B 0,C 180,E1 947.209,E2 947.209} C_VEL
LIN {X 0,Y 601.767,Z 370.16,A -85,B 0,C 180,E1 952.855,E2 952.855} C_VEL
LIN {X 0,Y 601.673,Z 370.16,A -85,B 0,C 180,E1 958.816,E2 958.816} C_VEL
LIN {X 0,Y 602.071,Z 370.16,A -85,B 0,C 180,E1 964.193,E2 964.193} C_VEL
LIN {X 0,Y 603.476,Z 397.923,A -85,B 0,C 180,E1 964.619,E2 964.619} C_VEL
LIN {X 0,Y 603.372,Z 442.114,A -85,B 0,C 180,E1 965.343,E2 965.343} C_VEL
LIN {X 0,Y 603.27,Z 478.436,A -85,B 0,C 180,E1 966.519,E2 966.519} C_VEL
LIN {X 0,Y 603.017,Z 511.947,A -85,B 0,C 180,E1 968.166,E2 968.166} C_VEL
LIN {X 0,Y 602.748,Z 544.534,A -85,B 0,C 180,E1 970.4,E2 970.4} C_VEL
LIN {X 0,Y 602.436,Z 572.822,A -85,B 0,C 180,E1 973.021,E2 973.021} C_VEL
LIN {X 0,Y 602.281,Z 596.971,A -85,B 0,C 180,E1 975.997,E2 975.997} C_VEL
LIN {X 0,Y 602.156,Z 616.349,A -85,B 0,C 180,E1 979.26,E2 979.26} C_VEL
LIN {X 0,Y 602.126,Z 629.454,A -85,B 0,C 180,E1 982.413,E2 982.413} C_VEL
LIN {X 0,Y 602.096,Z 637.967,A -85,B 0,C 180,E1 985.672,E2 985.672} C_VEL
LIN {X 0,Y 602.12,Z 641.506,A -85,B 0,C 180,E1 988.557,E2 988.557} C_VEL
LIN {X 0,Y 602.211,Z 641.509,A -85,B 0,C 180,E1 991.438,E2 991.438} C_VEL
LIN {X 0,Y 602.104,Z 636.457,A -85,B 0,C 180,E1 995.047,E2 995.047} C_VEL
LIN {X 0,Y 602.208,Z 626.847,A -85,B 0,C 180,E1 998.309,E2 998.309} C_VEL
LIN {X 0,Y 602.305,Z 610.846,A -85,B 0,C 180,E1 1001.782,E2 1001.782} C_VEL
LIN {X 0,Y 602.379,Z 589.202,A -85,B 0,C 180,E1 1005.056,E2 1005.056} C_VEL
LIN {X 0,Y 602.575,Z 563.538,A -85,B 0,C 180,E1 1007.923,E2 1007.923} C_VEL
LIN {X 0,Y 602.824,Z 532.906,A -85,B 0,C 180,E1 1010.48,E2 1010.48} C_VEL
LIN {X 0,Y 603.121,Z 500.433,A -85,B 0,C 180,E1 1012.466,E2 1012.466} C_VEL
LIN {X 0,Y 603.331,Z 465.637,A -85,B 0,C 180,E1 1013.963,E2 1013.963} C_VEL
LIN {X 0,Y 603.504,Z 428.294,A -85,B 0,C 180,E1 1014.949,E2 1014.949} C_VEL
LIN {X 0,Y 602.523,Z 372.336,A -85,B 0,C 180,E1 1015.755,E2 1015.755} C_VEL
LIN {X 0,Y 602.203,Z 370.16,A -85,B 0,C 180,E1 1015.848,E2 1015.848} C_VEL
LIN {X 0,Y 601.782,Z 370.16,A -85,B 0,C 180,E1 1021.889,E2 1021.889} C_VEL
LIN {X 0,Y 601.762,Z 370.16,A -85,B 0,C 180,E1 1027.14,E2 1027.14} C_VEL
LIN {X 0,Y 601.619,Z 370.16,A -85,B 0,C 180,E1 1032.797,E2 1032.797} C_VEL
LIN {X 0,Y 601.627,Z 370.16,A -85,B 0,C 180,E1 1039.015,E2 1039.015} C_VEL
LIN {X 0,Y 601.725,Z 370.16,A -85,B 0,C 180,E1 1044.642,E2 1044.642} C_VEL
LIN {X 0,Y 601.805,Z 370.16,A -85,B 0,C 180,E1 1049.792,E2 1049.792} C_VEL
LIN {X 0,Y 602.042,Z 370.16,A -85,B 0,C 180,E1 1054.855,E2 1054.855} C_VEL
LIN {X 0,Y 602.108,Z 370.16,A -85,B 0,C 180,E1 1059.337,E2 1059.337} C_VEL
LIN {X 0,Y 603.135,Z 405.108,A -85,B 0,C 180,E1 1060.039,E2 1060.039} C_VEL
LIN {X 0,Y 602.898,Z 437.9,A -85,B 0,C 180,E1 1061.232,E2 1061.232} C_VEL
LIN {X 0,Y 602.682,Z 468.27,A -85,B 0,C 180,E1 1062.933,E2 1062.933} C_VEL
LIN {X 0,Y 602.5,Z 496.279,A -85,B 0,C 180,E1 1065.16,E2 1065.16} C_VEL
LIN {X 0,Y 602.319,Z 520.481,A -85,B 0,C 180,E1 1067.847,E2 1067.847} C_VEL
LIN {X 0,Y 602.212,Z 538.09,A -85,B 0,C 180,E1 1070.595,E2 1070.595} C_VEL
LIN {X 0,Y 602.147,Z 551.73,A -85,B 0,C 180,E1 1073.729,E2 1073.729} C_VEL
LIN {X 0,Y 602.158,Z 558.688,A -85,B 0,C 180,E1 1076.395,E2 1076.395} C_VEL
LIN {X 0,Y 602.194,Z 561.45,A -85,B 0,C 180,E1 1078.558,E2 1078.558} C_VEL
LIN {X 0,Y 602.144,Z 561.389,A -85,B 0,C 180,E1 1081.44,E2 1081.44} C_VEL
LIN {X 0,Y 602.166,Z 556.981,A -85,B 0,C 180,E1 1084.325,E2 1084.325} C_VEL
LIN {X 0,Y 602.259,Z 546.383,A -85,B 0,C 180,E1 1087.582,E2 1087.582} C_VEL
LIN {X 0,Y 602.312,Z 530.478,A -85,B 0,C 180,E1 1090.622,E2 1090.622} C_VEL
LIN {X 0,Y 602.465,Z 509.08,A -85,B 0,C 180,E1 1093.44,E2 1093.44} C_VEL
LIN {X 0,Y 602.571,Z 483.549,A -85,B 0,C 180,E1 1095.855,E2 1095.855} C_VEL
LIN {X 0,Y 602.767,Z 454.589,A -85,B 0,C 180,E1 1097.823,E2 1097.823} C_VEL
LIN {X 0,Y 602.93,Z 422.135,A -85,B 0,C 180,E1 1099.333,E2 1099.333} C_VEL
LIN {X 0,Y 602.993,Z 386.726,A -85,B 0,C 180,E1 1100.297,E2 1100.297} C_VEL
LIN {X 0,Y 601.782,Z 370.16,A -85,B 0,C 180,E1 1100.621,E2 1100.621} C_VEL
LIN {X 0,Y 601.987,Z 370.16,A -85,B 0,C 180,E1 1105.309,E2 1105.309} C_VEL
LIN {X 0,Y 601.734,Z 370.16,A -85,B 0,C 180,E1 1111.198,E2 1111.198} C_VEL
LIN {X 0,Y 601.894,Z 370.16,A -85,B 0,C 180,E1 1117.131,E2 1117.131} C_VEL
LIN {X 0,Y 601.579,Z 370.16,A -85,B 0,C 180,E1 1122.801,E2 1122.801} C_VEL
LIN {X 0,Y 601.772,Z 370.16,A -85,B 0,C 180,E1 1127.217,E2 1127.217} C_VEL
LIN {X 0,Y 601.774,Z 370.16,A -85,B 0,C 180,E1 1132.861,E2 1132.861} C_VEL
LIN {X 0,Y 601.719,Z 370.16,A -85,B 0,C 180,E1 1138.805,E2 1138.805} C_VEL
LIN {X 0,Y 602.015,Z 370.16,A -85,B 0,C 180,E1 1144.862,E2 1144.862} C_VEL
LIN {X 0,Y 602.103,Z 370.181,A -85,B 0,C 180,E1 1149.339,E2 1149.339} C_VEL
LIN {X 0,Y 603.128,Z 406.521,A -85,B 0,C 180,E1 1150.08,E2 1150.08} C_VEL
LIN {X 0,Y 602.928,Z 439.012,A -85,B 0,C 180,E1 1151.283,E2 1151.283} C_VEL
LIN {X 0,Y 602.675,Z 470.068,A -85,B 0,C 180,E1 1153.055,E2 1153.055} C_VEL
LIN {X 0,Y 602.473,Z 497.773,A -85,B 0,C 180,E1 1155.305,E2 1155.305} C_VEL
LIN {X 0,Y 602.317,Z 520.507,A -85,B 0,C 180,E1 1157.85,E2 1157.85} C_VEL
LIN {X 0,Y 602.212,Z 538.104,A -85,B 0,C 180,E1 1160.598,E2 1160.598} C_VEL
LIN {X 0,Y 602.145,Z 551.737,A -85,B 0,C 180,E1 1163.732,E2 1163.732} C_VEL
LIN {X 0,Y 602.151,Z 558.694,A -85,B 0,C 180,E1 1166.398,E2 1166.398} C_VEL
LIN {X 0,Y 602.174,Z 561.449,A -85,B 0,C 180,E1 1168.562,E2 1168.562} C_VEL
LIN {X 0,Y 602.185,Z 561.383,A -85,B 0,C 180,E1 1171.443,E2 1171.443} C_VEL
LIN {X 0,Y 602.189,Z 556.971,A -85,B 0,C 180,E1 1174.328,E2 1174.328} C_VEL
LIN {X 0,Y 602.265,Z 546.364,A -85,B 0,C 180,E1 1177.586,E2 1177.586} C_VEL
LIN {X 0,Y 602.312,Z 530.455,A -85,B 0,C 180,E1 1180.625,E2 1180.625} C_VEL
LIN {X 0,Y 602.466,Z 509.051,A -85,B 0,C 180,E1 1183.443,E2 1183.443} C_VEL
LIN {X 0,Y 602.566,Z 483.497,A -85,B 0,C 180,E1 1185.859,E2 1185.859} C_VEL
LIN {X 0,Y 602.76,Z 454.511,A -85,B 0,C 180,E1 1187.827,E2 1187.827} C_VEL
LIN {X 0,Y 602.933,Z 422.038,A -85,B 0,C 180,E1 1189.336,E2 1189.336} C_VEL
LIN {X 0,Y 603.036,Z 388.884,A -85,B 0,C 180,E1 1190.252,E2 1190.252} C_VEL
LIN {X 0,Y 601.514,Z 370.16,A -85,B 0,C 180,E1 1190.634,E2 1190.634} C_VEL
LIN {X 0,Y 601.628,Z 370.16,A -85,B 0,C 180,E1 1195.33,E2 1195.33} C_VEL
LIN {X 0,Y 601.507,Z 370.16,A -85,B 0,C 180,E1 1200.226,E2 1200.226} C_VEL
LIN {X 0,Y 601.771,Z 370.16,A -85,B 0,C 180,E1 1203.883,E2 1203.883} C_VEL
LIN {X 0,Y 601.728,Z 370.16,A -85,B 0,C 180,E1 1208.979,E2 1208.979} C_VEL
LIN {X 0,Y 601.694,Z 370.16,A -85,B 0,C 180,E1 1215.212,E2 1215.212} C_VEL
LIN {X 0,Y 601.649,Z 370.16,A -85,B 0,C 180,E1 1221.02,E2 1221.02} C_VEL
LIN {X 0,Y 601.495,Z 370.16,A -85,B 0,C 180,E1 1226.163,E2 1226.163} C_VEL
LIN {X 0,Y 601.628,Z 370.16,A -85,B 0,C 180,E1 1231.439,E2 1231.439} C_VEL
LIN {X 0,Y 601.746,Z 370.16,A -85,B 0,C 180,E1 1236.264,E2 1236.264} C_VEL
LIN {X 0,Y 601.92,Z 370.16,A -85,B 0,C 180,E1 1240.916,E2 1240.916} C_VEL
LIN {X 0,Y 602.093,Z 370.16,A -85,B 0,C 180,E1 1246.922,E2 1246.922} C_VEL
LIN {X 0,Y 601.874,Z 370.16,A -85,B 0,C 180,E1 1252.776,E2 1252.776} C_VEL
LIN {X 0,Y 601.868,Z 370.16,A -85,B 0,C 180,E1 1257.667,E2 1257.667} C_VEL
LIN {X 0,Y 597.798,Z 370.16,A -85,B 0,C 180,E1 1259.291,E2 1259.291} C_VEL
LIN {X 0,Y 594.066,Z 370.16,A -85,B 0,C 180,E1 1260.937,E2 1260.937} C_VEL
LIN {X 0,Y 594.08,Z 370.16,A -85,B 0,C 180,E1 1266.333,E2 1266.333} C_VEL
LIN {X 0,Y 593.891,Z 370.16,A -85,B 0,C 180,E1 1271.768,E2 1271.768} C_VEL
LIN {X 0,Y 593.867,Z 370.16,A -85,B 0,C 180,E1 1276.286,E2 1276.286} C_VEL
LIN {X 0,Y 593.97,Z 370.16,A -85,B 0,C 180,E1 1280.907,E2 1280.907} C_VEL
LIN {X 0,Y 593.924,Z 370.16,A -85,B 0,C 180,E1 1285.68,E2 1285.68} C_VEL
LIN {X 0,Y 593.836,Z 370.16,A -85,B 0,C 180,E1 1290.657,E2 1290.657} C_VEL
LIN {X 0,Y 593.893,Z 370.16,A -85,B 0,C 180,E1 1295.896,E2 1295.896} C_VEL
LIN {X 0,Y 593.632,Z 370.16,A -85,B 0,C 180,E1 1301.535,E2 1301.535} C_VEL
LIN {X 0,Y 593.797,Z 370.16,A -85,B 0,C 180,E1 1306.495,E2 1306.495} C_VEL
LIN {X 0,Y 593.799,Z 370.16,A -85,B 0,C 180,E1 1312.271,E2 1312.271} C_VEL
LIN {X 0,Y 593.6,Z 370.16,A -85,B 0,C 180,E1 1317.614,E2 1317.614} C_VEL
LIN {X 0,Y 593.85,Z 370.16,A -85,B 0,C 180,E1 1323.16,E2 1323.16} C_VEL
LIN {X 0,Y 594.023,Z 370.16,A -85,B 0,C 180,E1 1323.787,E2 1323.787} C_VEL
LIN {X 0,Y 596.086,Z 379.36,A -85,B 0,C 180,E1 1324.038,E2 1324.038} C_VEL
LIN {X 0,Y 596.192,Z 439.638,A -85,B 0,C 180,E1 1324.963,E2 1324.963} C_VEL
LIN {X 0,Y 595.965,Z 476.57,A -85,B 0,C 180,E1 1326.136,E2 1326.136} C_VEL
LIN {X 0,Y 595.575,Z 510.398,A -85,B 0,C 180,E1 1327.788,E2 1327.788} C_VEL
LIN {X 0,Y 595.184,Z 543.087,A -85,B 0,C 180,E1 1330.023,E2 1330.023} C_VEL
LIN {X 0,Y 594.748,Z 572.591,A -85,B 0,C 180,E1 1332.769,E2 1332.769} C_VEL
LIN {X 0,Y 594.501,Z 596.395,A -85,B 0,C 180,E1 1335.728,E2 1335.728} C_VEL
LIN {X 0,Y 594.331,Z 615.416,A -85,B 0,C 180,E1 1338.926,E2 1338.926} C_VEL
LIN {X 0,Y 594.251,Z 629.454,A -85,B 0,C 180,E1 1342.311,E2 1342.311} C_VEL
LIN {X 0,Y 594.198,Z 637.966,A -85,B 0,C 180,E1 1345.614,E2 1345.614} C_VEL
LIN {X 0,Y 594.218,Z 641.506,A -85,B 0,C 180,E1 1348.538,E2 1348.538} C_VEL
LIN {X 0,Y 594.306,Z 641.509,A -85,B 0,C 180,E1 1351.458,E2 1351.458} C_VEL
LIN {X 0,Y 594.233,Z 636.458,A -85,B 0,C 180,E1 1355.114,E2 1355.114} C_VEL
LIN {X 0,Y 594.309,Z 626.847,A -85,B 0,C 180,E1 1358.42,E2 1358.42} C_VEL
LIN {X 0,Y 594.432,Z 610.847,A -85,B 0,C 180,E1 1361.94,E2 1361.94} C_VEL
LIN {X 0,Y 594.581,Z 590.226,A -85,B 0,C 180,E1 1365.126,E2 1365.126} C_VEL
LIN {X 0,Y 594.874,Z 565.454,A -85,B 0,C 180,E1 1367.971,E2 1367.971} C_VEL
LIN {X 0,Y 595.272,Z 534.834,A -85,B 0,C 180,E1 1370.613,E2 1370.613} C_VEL
LIN {X 0,Y 595.718,Z 502.035,A -85,B 0,C 180,E1 1372.677,E2 1372.677} C_VEL
LIN {X 0,Y 596.05,Z 467.541,A -85,B 0,C 180,E1 1374.207,E2 1374.207} C_VEL
LIN {X 0,Y 596.285,Z 430.999,A -85,B 0,C 180,E1 1375.217,E2 1375.217} C_VEL
LIN {X 0,Y 595.614,Z 374.594,A -85,B 0,C 180,E1 1376.047,E2 1376.047} C_VEL
LIN {X 0,Y 594.254,Z 370.16,A -85,B 0,C 180,E1 1376.28,E2 1376.28} C_VEL
LIN {X 0,Y 593.924,Z 370.16,A -85,B 0,C 180,E1 1382.735,E2 1382.735} C_VEL
LIN {X 0,Y 593.792,Z 370.16,A -85,B 0,C 180,E1 1387.779,E2 1387.779} C_VEL
LIN {X 0,Y 593.595,Z 370.16,A -85,B 0,C 180,E1 1393.518,E2 1393.518} C_VEL
LIN {X 0,Y 593.677,Z 370.16,A -85,B 0,C 180,E1 1398.469,E2 1398.469} C_VEL
LIN {X 0,Y 593.832,Z 370.16,A -85,B 0,C 180,E1 1404.664,E2 1404.664} C_VEL
LIN {X 0,Y 593.769,Z 370.16,A -85,B 0,C 180,E1 1411.024,E2 1411.024} C_VEL
LIN {X 0,Y 593.901,Z 370.16,A -85,B 0,C 180,E1 1415.929,E2 1415.929} C_VEL
LIN {X 0,Y 594.106,Z 370.16,A -85,B 0,C 180,E1 1419.037,E2 1419.037} C_VEL
LIN {X 0,Y 595.559,Z 381.703,A -85,B 0,C 180,E1 1419.264,E2 1419.264} C_VEL
LIN {X 0,Y 595.576,Z 415.488,A -85,B 0,C 180,E1 1420.097,E2 1420.097} C_VEL
LIN {X 0,Y 595.291,Z 447.573,A -85,B 0,C 180,E1 1421.464,E2 1421.464} C_VEL
LIN {X 0,Y 594.957,Z 476.708,A -85,B 0,C 180,E1 1423.309,E2 1423.309} C_VEL
LIN {X 0,Y 594.694,Z 503.34,A -85,B 0,C 180,E1 1425.667,E2 1425.667} C_VEL
LIN {X 0,Y 594.527,Z 525.724,A -85,B 0,C 180,E1 1428.422,E2 1428.422} C_VEL
LIN {X 0,Y 594.339,Z 541.835,A -85,B 0,C 180,E1 1431.208,E2 1431.208} C_VEL
LIN {X 0,Y 594.273,Z 553.304,A -85,B 0,C 180,E1 1434.15,E2 1434.15} C_VEL
LIN {X 0,Y 594.215,Z 559.872,A -85,B 0,C 180,E1 1437.078,E2 1437.078} C_VEL
LIN {X 0,Y 594.207,Z 561.998,A -85,B 0,C 180,E1 1439.999,E2 1439.999} C_VEL
LIN {X 0,Y 594.217,Z 559.732,A -85,B 0,C 180,E1 1442.92,E2 1442.92} C_VEL
LIN {X 0,Y 594.311,Z 553.023,A -85,B 0,C 180,E1 1445.847,E2 1445.847} C_VEL
LIN {X 0,Y 594.346,Z 541.417,A -85,B 0,C 180,E1 1448.79,E2 1448.79} C_VEL
LIN {X 0,Y 594.532,Z 523.863,A -85,B 0,C 180,E1 1451.753,E2 1451.753} C_VEL
LIN {X 0,Y 594.708,Z 501.451,A -85,B 0,C 180,E1 1454.436,E2 1454.436} C_VEL
LIN {X 0,Y 595.013,Z 473.587,A -85,B 0,C 180,E1 1456.834,E2 1456.834} C_VEL
LIN {X 0,Y 595.349,Z 442.095,A -85,B 0,C 180,E1 1458.725,E2 1458.725} C_VEL
LIN {X 0,Y 595.643,Z 409.944,A -85,B 0,C 180,E1 1459.99,E2 1459.99} C_VEL
LIN {X 0,Y 594.877,Z 374.274,A -85,B 0,C 180,E1 1460.781,E2 1460.781} C_VEL
LIN {X 0,Y 593.857,Z 370.16,A -85,B 0,C 180,E1 1460.909,E2 1460.909} C_VEL
LIN {X 0,Y 593.972,Z 370.16,A -85,B 0,C 180,E1 1465.676,E2 1465.676} C_VEL
LIN {X 0,Y 593.872,Z 370.16,A -85,B 0,C 180,E1 1470.652,E2 1470.652} C_VEL
LIN {X 0,Y 593.908,Z 370.16,A -85,B 0,C 180,E1 1475.893,E2 1475.893} C_VEL
LIN {X 0,Y 593.641,Z 370.16,A -85,B 0,C 180,E1 1481.532,E2 1481.532} C_VEL
LIN {X 0,Y 593.805,Z 370.16,A -85,B 0,C 180,E1 1486.501,E2 1486.501} C_VEL
LIN {X 0,Y 593.806,Z 370.16,A -85,B 0,C 180,E1 1492.277,E2 1492.277} C_VEL
LIN {X 0,Y 593.655,Z 370.16,A -85,B 0,C 180,E1 1497.622,E2 1497.622} C_VEL
LIN {X 0,Y 593.727,Z 370.16,A -85,B 0,C 180,E1 1502.681,E2 1502.681} C_VEL
LIN {X 0,Y 593.89,Z 370.16,A -85,B 0,C 180,E1 1508.311,E2 1508.311} C_VEL
LIN {X 0,Y 594.105,Z 370.16,A -85,B 0,C 180,E1 1509.028,E2 1509.028} C_VEL
LIN {X 0,Y 595.543,Z 382.668,A -85,B 0,C 180,E1 1509.277,E2 1509.277} C_VEL
LIN {X 0,Y 595.517,Z 418.008,A -85,B 0,C 180,E1 1510.182,E2 1510.182} C_VEL
LIN {X 0,Y 595.186,Z 451.125,A -85,B 0,C 180,E1 1511.655,E2 1511.655} C_VEL
LIN {X 0,Y 594.939,Z 480.553,A -85,B 0,C 180,E1 1513.602,E2 1513.602} C_VEL
LIN {X 0,Y 594.685,Z 506.758,A -85,B 0,C 180,E1 1516.035,E2 1516.035} C_VEL
LIN {X 0,Y 594.506,Z 528.606,A -85,B 0,C 180,E1 1518.859,E2 1518.859} C_VEL
LIN {X 0,Y 594.378,Z 545.225,A -85,B 0,C 180,E1 1521.949,E2 1521.949} C_VEL
LIN {X 0,Y 594.33,Z 555.379,A -85,B 0,C 180,E1 1524.887,E2 1524.887} C_VEL
LIN {X 0,Y 594.208,Z 559.886,A -85,B 0,C 180,E1 1527.081,E2 1527.081} C_VEL
LIN {X 0,Y 594.217,Z 561.996,A -85,B 0,C 180,E1 1530.002,E2 1530.002} C_VEL
LIN {X 0,Y 594.24,Z 559.732,A -85,B 0,C 180,E1 1532.923,E2 1532.923} C_VEL
LIN {X 0,Y 594.327,Z 553.014,A -85,B 0,C 180,E1 1535.85,E2 1535.85} C_VEL
LIN {X 0,Y 594.348,Z 541.394,A -85,B 0,C 180,E1 1538.793,E2 1538.793} C_VEL
LIN {X 0,Y 594.536,Z 523.834,A -85,B 0,C 180,E1 1541.756,E2 1541.756} C_VEL
LIN {X 0,Y 594.734,Z 501.462,A -85,B 0,C 180,E1 1544.437,E2 1544.437} C_VEL
LIN {X 0,Y 594.998,Z 475.504,A -85,B 0,C 180,E1 1546.69,E2 1546.69} C_VEL
LIN {X 0,Y 595.267,Z 445.76,A -85,B 0,C 180,E1 1548.539,E2 1548.539} C_VEL
LIN {X 0,Y 595.587,Z 412.592,A -85,B 0,C 180,E1 1549.912,E2 1549.912} C_VEL
LIN {X 0,Y 595.142,Z 376.943,A -85,B 0,C 180,E1 1550.734,E2 1550.734} C_VEL
LIN {X 0,Y 593.703,Z 370.16,A -85,B 0,C 180,E1 1550.918,E2 1550.918} C_VEL
LIN {X 0,Y 593.717,Z 370.16,A -85,B 0,C 180,E1 1555.691,E2 1555.691} C_VEL
LIN {X 0,Y 593.612,Z 370.16,A -85,B 0,C 180,E1 1560.671,E2 1560.671} C_VEL
LIN {X 0,Y 593.652,Z 370.16,A -85,B 0,C 180,E1 1565.31,E2 1565.31} C_VEL
LIN {X 0,Y 593.645,Z 370.16,A -85,B 0,C 180,E1 1570.089,E2 1570.089} C_VEL
LIN {X 0,Y 593.763,Z 370.16,A -85,B 0,C 180,E1 1575.558,E2 1575.558} C_VEL
LIN {X 0,Y 593.693,Z 370.16,A -85,B 0,C 180,E1 1580.396,E2 1580.396} C_VEL
LIN {X 0,Y 593.608,Z 370.16,A -85,B 0,C 180,E1 1585.871,E2 1585.871} C_VEL
LIN {X 0,Y 593.715,Z 370.16,A -85,B 0,C 180,E1 1591.023,E2 1591.023} C_VEL
LIN {X 0,Y 593.908,Z 370.16,A -85,B 0,C 180,E1 1595.931,E2 1595.931} C_VEL
LIN {X 0,Y 593.991,Z 370.16,A -85,B 0,C 180,E1 1600.651,E2 1600.651} C_VEL
LIN {X 0,Y 594.154,Z 370.16,A -85,B 0,C 180,E1 1606.744,E2 1606.744} C_VEL
LIN {X 0,Y 593.98,Z 370.16,A -85,B 0,C 180,E1 1612.679,E2 1612.679} C_VEL
LIN {X 0,Y 593.961,Z 370.16,A -85,B 0,C 180,E1 1617.651,E2 1617.651} C_VEL
LIN {X 0,Y 594.066,Z 370.16,A -85,B 0,C 180,E1 1620.937,E2 1620.937} C_VEL
LIN {X 0,Y 591.558,Z 370.16,A -85,B 0,C 180,E1 1622.181,E2 1622.181} C_VEL
LIN {X 0,Y 586.066,Z 370.16,A -85,B 0,C 180,E1 1624.041,E2 1624.041} C_VEL
LIN {X 0,Y 585.993,Z 370.16,A -85,B 0,C 180,E1 1624.256,E2 1624.256} C_VEL
LIN {X 0,Y 585.931,Z 370.16,A -85,B 0,C 180,E1 1628.919,E2 1628.919} C_VEL
LIN {X 0,Y 585.924,Z 370.16,A -85,B 0,C 180,E1 1633.448,E2 1633.448} C_VEL
LIN {X 0,Y 586.034,Z 370.16,A -85,B 0,C 180,E1 1639.624,E2 1639.624} C_VEL
LIN {X 0,Y 585.958,Z 370.16,A -85,B 0,C 180,E1 1646.055,E2 1646.055} C_VEL
LIN {X 0,Y 585.789,Z 370.16,A -85,B 0,C 180,E1 1651.472,E2 1651.472} C_VEL
LIN {X 0,Y 585.955,Z 370.16,A -85,B 0,C 180,E1 1656.776,E2 1656.776} C_VEL
LIN {X 0,Y 585.732,Z 370.16,A -85,B 0,C 180,E1 1662.223,E2 1662.223} C_VEL
LIN {X 0,Y 585.878,Z 370.16,A -85,B 0,C 180,E1 1667.787,E2 1667.787} C_VEL
LIN {X 0,Y 585.866,Z 370.16,A -85,B 0,C 180,E1 1673.532,E2 1673.532} C_VEL
LIN {X 0,Y 585.807,Z 370.16,A -85,B 0,C 180,E1 1678.875,E2 1678.875} C_VEL
LIN {X 0,Y 586.025,Z 370.16,A -85,B 0,C 180,E1 1683.402,E2 1683.402} C_VEL
LIN {X 0,Y 588.949,Z 379.402,A -85,B 0,C 180,E1 1683.7,E2 1683.7} C_VEL
LIN {X 0,Y 589.019,Z 440.169,A -85,B 0,C 180,E1 1684.651,E2 1684.651} C_VEL
LIN {X 0,Y 588.694,Z 476.572,A -85,B 0,C 180,E1 1685.823,E2 1685.823} C_VEL
LIN {X 0,Y 588.134,Z 510.481,A -85,B 0,C 180,E1 1687.497,E2 1687.497} C_VEL
LIN {X 0,Y 587.595,Z 542.568,A -85,B 0,C 180,E1 1689.713,E2 1689.713} C_VEL
LIN {X 0,Y 587.068,Z 572.038,A -85,B 0,C 180,E1 1692.476,E2 1692.476} C_VEL
LIN {X 0,Y 586.717,Z 596.071,A -85,B 0,C 180,E1 1695.489,E2 1695.489} C_VEL
LIN {X 0,Y 586.481,Z 615.496,A -85,B 0,C 180,E1 1698.791,E2 1698.791} C_VEL
LIN {X 0,Y 586.38,Z 629.454,A -85,B 0,C 180,E1 1702.208,E2 1702.208} C_VEL
LIN {X 0,Y 586.303,Z 637.966,A -85,B 0,C 180,E1 1705.555,E2 1705.555} C_VEL
LIN {X 0,Y 586.321,Z 641.506,A -85,B 0,C 180,E1 1708.518,E2 1708.518} C_VEL
LIN {X 0,Y 586.402,Z 641.509,A -85,B 0,C 180,E1 1711.477,E2 1711.477} C_VEL
LIN {X 0,Y 586.349,Z 636.458,A -85,B 0,C 180,E1 1715.183,E2 1715.183} C_VEL
LIN {X 0,Y 586.406,Z 625.507,A -85,B 0,C 180,E1 1718.909,E2 1718.909} C_VEL
LIN {X 0,Y 586.567,Z 609.819,A -85,B 0,C 180,E1 1722.292,E2 1722.292} C_VEL
LIN {X 0,Y 586.805,Z 588.761,A -85,B 0,C 180,E1 1725.523,E2 1725.523} C_VEL
LIN {X 0,Y 587.235,Z 563.538,A -85,B 0,C 180,E1 1728.408,E2 1728.408} C_VEL
LIN {X 0,Y 587.754,Z 533.425,A -85,B 0,C 180,E1 1730.992,E2 1730.992} C_VEL
LIN {X 0,Y 588.327,Z 499.949,A -85,B 0,C 180,E1 1733.089,E2 1733.089} C_VEL
LIN {X 0,Y 588.84,Z 465.643,A -85,B 0,C 180,E1 1734.592,E2 1734.592} C_VEL
LIN {X 0,Y 589.188,Z 429.432,A -85,B 0,C 180,E1 1735.575,E2 1735.575} C_VEL
LIN {X 0,Y 588.359,Z 376.684,A -85,B 0,C 180,E1 1736.364,E2 1736.364} C_VEL
LIN {X 0,Y 586.324,Z 370.16,A -85,B 0,C 180,E1 1736.58,E2 1736.58} C_VEL
LIN {X 0,Y 586.024,Z 370.16,A -85,B 0,C 180,E1 1742.852,E2 1742.852} C_VEL
LIN {X 0,Y 585.825,Z 370.16,A -85,B 0,C 180,E1 1748.33,E2 1748.33} C_VEL
LIN {X 0,Y 585.709,Z 370.16,A -85,B 0,C 180,E1 1753.636,E2 1753.636} C_VEL
LIN {X 0,Y 585.762,Z 370.16,A -85,B 0,C 180,E1 1758.545,E2 1758.545} C_VEL
LIN {X 0,Y 585.799,Z 370.16,A -85,B 0,C 180,E1 1763.529,E2 1763.529} C_VEL
LIN {X 0,Y 585.858,Z 370.16,A -85,B 0,C 180,E1 1768.88,E2 1768.88} C_VEL
LIN {X 0,Y 586.019,Z 370.16,A -85,B 0,C 180,E1 1774.71,E2 1774.71} C_VEL
LIN {X 0,Y 586.173,Z 370.916,A -85,B 0,C 180,E1 1778.762,E2 1778.762} C_VEL
LIN {X 0,Y 588.193,Z 382.418,A -85,B 0,C 180,E1 1779.005,E2 1779.005} C_VEL
LIN {X 0,Y 588.088,Z 416.91,A -85,B 0,C 180,E1 1779.884,E2 1779.884} C_VEL
LIN {X 0,Y 587.754,Z 447.548,A -85,B 0,C 180,E1 1781.217,E2 1781.217} C_VEL
LIN {X 0,Y 587.286,Z 477.197,A -85,B 0,C 180,E1 1783.122,E2 1783.122} C_VEL
LIN {X 0,Y 586.933,Z 504.428,A -85,B 0,C 180,E1 1785.591,E2 1785.591} C_VEL
LIN {X 0,Y 586.694,Z 527.061,A -85,B 0,C 180,E1 1788.467,E2 1788.467} C_VEL
LIN {X 0,Y 586.522,Z 543.58,A -85,B 0,C 180,E1 1791.464,E2 1791.464} C_VEL
LIN {X 0,Y 586.443,Z 555.382,A -85,B 0,C 180,E1 1794.815,E2 1794.815} C_VEL
LIN {X 0,Y 586.321,Z 559.866,A -85,B 0,C 180,E1 1797.039,E2 1797.039} C_VEL
LIN {X 0,Y 586.308,Z 561.999,A -85,B 0,C 180,E1 1799.999,E2 1799.999} C_VEL
LIN {X 0,Y 586.321,Z 559.732,A -85,B 0,C 180,E1 1802.959,E2 1802.959} C_VEL
LIN {X 0,Y 586.4,Z 551.925,A -85,B 0,C 180,E1 1806.284,E2 1806.284} C_VEL
LIN {X 0,Y 586.489,Z 539.564,A -85,B 0,C 180,E1 1809.283,E2 1809.283} C_VEL
LIN {X 0,Y 586.662,Z 521.202,A -85,B 0,C 180,E1 1812.291,E2 1812.291} C_VEL
LIN {X 0,Y 586.998,Z 498.322,A -85,B 0,C 180,E1 1814.945,E2 1814.945} C_VEL
LIN {X 0,Y 587.402,Z 471.7,A -85,B 0,C 180,E1 1817.192,E2 1817.192} C_VEL
LIN {X 0,Y 587.859,Z 441.12,A -85,B 0,C 180,E1 1819.021,E2 1819.021} C_VEL
LIN {X 0,Y 588.194,Z 408.339,A -85,B 0,C 180,E1 1820.304,E2 1820.304} C_VEL
LIN {X 0,Y 587.326,Z 375.58,A -85,B 0,C 180,E1 1821.044,E2 1821.044} C_VEL
LIN {X 0,Y 585.906,Z 370.16,A -85,B 0,C 180,E1 1821.206,E2 1821.206} C_VEL
LIN {X 0,Y 586.001,Z 370.16,A -85,B 0,C 180,E1 1826.051,E2 1826.051} C_VEL
LIN {X 0,Y 585.827,Z 370.16,A -85,B 0,C 180,E1 1831.486,E2 1831.486} C_VEL
LIN {X 0,Y 585.973,Z 370.16,A -85,B 0,C 180,E1 1836.786,E2 1836.786} C_VEL
LIN {X 0,Y 585.732,Z 370.16,A -85,B 0,C 180,E1 1842.221,E2 1842.221} C_VEL
LIN {X 0,Y 585.897,Z 370.16,A -85,B 0,C 180,E1 1847.795,E2 1847.795} C_VEL
LIN {X 0,Y 585.863,Z 370.16,A -85,B 0,C 180,E1 1853.537,E2 1853.537} C_VEL
LIN {X 0,Y 585.847,Z 370.16,A -85,B 0,C 180,E1 1858.882,E2 1858.882} C_VEL
LIN {X 0,Y 586.012,Z 370.16,A -85,B 0,C 180,E1 1864.712,E2 1864.712} C_VEL
LIN {X 0,Y 586.107,Z 370.16,A -85,B 0,C 180,E1 1868.733,E2 1868.733} C_VEL
LIN {X 0,Y 588.142,Z 382.7,A -85,B 0,C 180,E1 1869.005,E2 1869.005} C_VEL
LIN {X 0,Y 588.099,Z 416.863,A -85,B 0,C 180,E1 1869.881,E2 1869.881} C_VEL
LIN {X 0,Y 587.667,Z 449.405,A -85,B 0,C 180,E1 1871.315,E2 1871.315} C_VEL
LIN {X 0,Y 587.282,Z 478.982,A -85,B 0,C 180,E1 1873.261,E2 1873.261} C_VEL
LIN {X 0,Y 586.932,Z 504.423,A -85,B 0,C 180,E1 1875.593,E2 1875.593} C_VEL
LIN {X 0,Y 586.686,Z 525.837,A -85,B 0,C 180,E1 1878.279,E2 1878.279} C_VEL
LIN {X 0,Y 586.468,Z 541.837,A -85,B 0,C 180,E1 1881.092,E2 1881.092} C_VEL
LIN {X 0,Y 586.368,Z 553.306,A -85,B 0,C 180,E1 1884.074,E2 1884.074} C_VEL
LIN {X 0,Y 586.314,Z 559.886,A -85,B 0,C 180,E1 1887.042,E2 1887.042} C_VEL
LIN {X 0,Y 586.317,Z 561.996,A -85,B 0,C 180,E1 1890.002,E2 1890.002} C_VEL
LIN {X 0,Y 586.342,Z 559.734,A -85,B 0,C 180,E1 1892.962,E2 1892.962} C_VEL
LIN {X 0,Y 586.414,Z 551.91,A -85,B 0,C 180,E1 1896.289,E2 1896.289} C_VEL
LIN {X 0,Y 586.492,Z 539.561,A -85,B 0,C 180,E1 1899.287,E2 1899.287} C_VEL
LIN {X 0,Y 586.666,Z 521.171,A -85,B 0,C 180,E1 1902.294,E2 1902.294} C_VEL
LIN {X 0,Y 587.007,Z 498.296,A -85,B 0,C 180,E1 1904.948,E2 1904.948} C_VEL
LIN {X 0,Y 587.443,Z 470.417,A -85,B 0,C 180,E1 1907.283,E2 1907.283} C_VEL
LIN {X 0,Y 587.861,Z 439.052,A -85,B 0,C 180,E1 1909.122,E2 1909.122} C_VEL
LIN {X 0,Y 588.223,Z 406.898,A -85,B 0,C 180,E1 1910.344,E2 1910.344} C_VEL
LIN {X 0,Y 587.197,Z 375.74,A -85,B 0,C 180,E1 1911.046,E2 1911.046} C_VEL
LIN {X 0,Y 585.813,Z 370.16,A -85,B 0,C 180,E1 1911.213,E2 1911.213} C_VEL
LIN {X 0,Y 585.846,Z 370.16,A -85,B 0,C 180,E1 1916.062,E2 1916.062} C_VEL
LIN {X 0,Y 585.734,Z 370.16,A -85,B 0,C 180,E1 1921.47,E2 1921.47} C_VEL
LIN {X 0,Y 585.636,Z 370.16,A -85,B 0,C 180,E1 1926.485,E2 1926.485} C_VEL
LIN {X 0,Y 585.683,Z 370.16,A -85,B 0,C 180,E1 1931.445,E2 1931.445} C_VEL
LIN {X 0,Y 585.889,Z 370.16,A -85,B 0,C 180,E1 1936.349,E2 1936.349} C_VEL
LIN {X 0,Y 585.765,Z 370.16,A -85,B 0,C 180,E1 1941.665,E2 1941.665} C_VEL
LIN {X 0,Y 585.674,Z 370.16,A -85,B 0,C 180,E1 1947.125,E2 1947.125} C_VEL
LIN {X 0,Y 585.769,Z 370.16,A -85,B 0,C 180,E1 1952.278,E2 1952.278} C_VEL
LIN {X 0,Y 585.858,Z 370.16,A -85,B 0,C 180,E1 1957.195,E2 1957.195} C_VEL
LIN {X 0,Y 586.013,Z 370.16,A -85,B 0,C 180,E1 1961.941,E2 1961.941} C_VEL
LIN {X 0,Y 586.23,Z 370.16,A -85,B 0,C 180,E1 1966.561,E2 1966.561} C_VEL
LIN {X 0,Y 586.076,Z 370.16,A -85,B 0,C 180,E1 1972.58,E2 1972.58} C_VEL
LIN {X 0,Y 586.218,Z 370.16,A -85,B 0,C 180,E1 1977.04,E2 1977.04} C_VEL
LIN {X 0,Y 586.289,Z 370.16,A -85,B 0,C 180,E1 1981.481,E2 1981.481} C_VEL
LIN {X 0,Y 585.993,Z 370.16,A -85,B 0,C 180,E1 1984.256,E2 1984.256} C_VEL
LIN {X 0,Y 583.568,Z 370.16,A -85,B 0,C 180,E1 1985.519,E2 1985.519} C_VEL
LIN {X 0,Y 578.045,Z 370.16,A -85,B 0,C 180,E1 1987.628,E2 1987.628} C_VEL
LIN {X 0,Y 578.058,Z 370.16,A -85,B 0,C 180,E1 1992.095,E2 1992.095} C_VEL
LIN {X 0,Y 578.01,Z 370.16,A -85,B 0,C 180,E1 1996.746,E2 1996.746} C_VEL
LIN {X 0,Y 578.054,Z 370.16,A -85,B 0,C 180,E1 2001.511,E2 2001.511} C_VEL
LIN {X 0,Y 577.899,Z 370.16,A -85,B 0,C 180,E1 2007.034,E2 2007.034} C_VEL
LIN {X 0,Y 577.882,Z 370.16,A -85,B 0,C 180,E1 2011.599,E2 2011.599} C_VEL
LIN {X 0,Y 578.041,Z 370.16,A -85,B 0,C 180,E1 2017.042,E2 2017.042} C_VEL
LIN {X 0,Y 577.86,Z 370.16,A -85,B 0,C 180,E1 2022.936,E2 2022.936} C_VEL
LIN {X 0,Y 577.942,Z 370.16,A -85,B 0,C 180,E1 2027.178,E2 2027.178} C_VEL
LIN {X 0,Y 577.949,Z 370.16,A -85,B 0,C 180,E1 2032.949,E2 2032.949} C_VEL
LIN {X 0,Y 577.866,Z 370.16,A -85,B 0,C 180,E1 2038.398,E2 2038.398} C_VEL
LIN {X 0,Y 578.034,Z 370.16,A -85,B 0,C 180,E1 2043.027,E2 2043.027} C_VEL
LIN {X 0,Y 581.979,Z 382.016,A -85,B 0,C 180,E1 2043.396,E2 2043.396} C_VEL
LIN {X 0,Y 581.873,Z 439.937,A -85,B 0,C 180,E1 2044.311,E2 2044.311} C_VEL
LIN {X 0,Y 581.428,Z 476.954,A -85,B 0,C 180,E1 2045.517,E2 2045.517} C_VEL
LIN {X 0,Y 580.723,Z 510.481,A -85,B 0,C 180,E1 2047.193,E2 2047.193} C_VEL
LIN {X 0,Y 580.029,Z 542.947,A -85,B 0,C 180,E1 2049.466,E2 2049.466} C_VEL
LIN {X 0,Y 579.384,Z 572.036,A -85,B 0,C 180,E1 2052.235,E2 2052.235} C_VEL
LIN {X 0,Y 578.927,Z 596.624,A -85,B 0,C 180,E1 2055.369,E2 2055.369} C_VEL
LIN {X 0,Y 578.627,Z 615.495,A -85,B 0,C 180,E1 2058.637,E2 2058.637} C_VEL
LIN {X 0,Y 578.52,Z 629.454,A -85,B 0,C 180,E1 2062.101,E2 2062.101} C_VEL
LIN {X 0,Y 578.409,Z 637.965,A -85,B 0,C 180,E1 2065.494,E2 2065.494} C_VEL
LIN {X 0,Y 578.419,Z 641.507,A -85,B 0,C 180,E1 2068.498,E2 2068.498} C_VEL
LIN {X 0,Y 578.497,Z 641.51,A -85,B 0,C 180,E1 2071.497,E2 2071.497} C_VEL
LIN {X 0,Y 578.463,Z 636.494,A -85,B 0,C 180,E1 2075.237,E2 2075.237} C_VEL
LIN {X 0,Y 578.535,Z 626.846,A -85,B 0,C 180,E1 2078.652,E2 2078.652} C_VEL
LIN {X 0,Y 578.709,Z 610.849,A -85,B 0,C 180,E1 2082.27,E2 2082.27} C_VEL
LIN {X 0,Y 579.031,Z 590.223,A -85,B 0,C 180,E1 2085.543,E2 2085.543} C_VEL
LIN {X 0,Y 579.514,Z 565.453,A -85,B 0,C 180,E1 2088.464,E2 2088.464} C_VEL
LIN {X 0,Y 580.178,Z 535.849,A -85,B 0,C 180,E1 2091.094,E2 2091.094} C_VEL
LIN {X 0,Y 580.969,Z 502.767,A -85,B 0,C 180,E1 2093.247,E2 2093.247} C_VEL
LIN {X 0,Y 581.559,Z 468.275,A -85,B 0,C 180,E1 2094.823,E2 2094.823} C_VEL
LIN {X 0,Y 582.018,Z 431.889,A -85,B 0,C 180,E1 2095.861,E2 2095.861} C_VEL
LIN {X 0,Y 581.462,Z 379.143,A -85,B 0,C 180,E1 2096.668,E2 2096.668} C_VEL
LIN {X 0,Y 578.335,Z 370.16,A -85,B 0,C 180,E1 2096.999,E2 2096.999} C_VEL
LIN {X 0,Y 578.109,Z 370.16,A -85,B 0,C 180,E1 2103.36,E2 2103.36} C_VEL
LIN {X 0,Y 577.901,Z 370.16,A -85,B 0,C 180,E1 2108.954,E2 2108.954} C_VEL
LIN {X 0,Y 577.725,Z 370.16,A -85,B 0,C 180,E1 2114.965,E2 2114.965} C_VEL
LIN {X 0,Y 577.793,Z 370.16,A -85,B 0,C 180,E1 2119.448,E2 2119.448} C_VEL
LIN {X 0,Y 577.851,Z 370.16,A -85,B 0,C 180,E1 2124.803,E2 2124.803} C_VEL
LIN {X 0,Y 577.938,Z 370.16,A -85,B 0,C 180,E1 2130.151,E2 2130.151} C_VEL
LIN {X 0,Y 578.095,Z 370.16,A -85,B 0,C 180,E1 2135.227,E2 2135.227} C_VEL
LIN {X 0,Y 578.156,Z 370.16,A -85,B 0,C 180,E1 2138.435,E2 2138.435} C_VEL
LIN {X 0,Y 580.817,Z 382.927,A -85,B 0,C 180,E1 2138.735,E2 2138.735} C_VEL
LIN {X 0,Y 580.678,Z 416.46,A -85,B 0,C 180,E1 2139.601,E2 2139.601} C_VEL
LIN {X 0,Y 580.203,Z 447.518,A -85,B 0,C 180,E1 2140.963,E2 2140.963} C_VEL
LIN {X 0,Y 579.628,Z 478.055,A -85,B 0,C 180,E1 2142.96,E2 2142.96} C_VEL
LIN {X 0,Y 579.162,Z 504.654,A -85,B 0,C 180,E1 2145.419,E2 2145.419} C_VEL
LIN {X 0,Y 578.858,Z 527.043,A -85,B 0,C 180,E1 2148.308,E2 2148.308} C_VEL
LIN {X 0,Y 578.635,Z 543.582,A -85,B 0,C 180,E1 2151.347,E2 2151.347} C_VEL
LIN {X 0,Y 578.557,Z 555.385,A -85,B 0,C 180,E1 2154.744,E2 2154.744} C_VEL
LIN {X 0,Y 578.423,Z 559.859,A -85,B 0,C 180,E1 2156.998,E2 2156.998} C_VEL
LIN {X 0,Y 578.409,Z 561.999,A -85,B 0,C 180,E1 2159.999,E2 2159.999} C_VEL
LIN {X 0,Y 578.421,Z 559.732,A -85,B 0,C 180,E1 2163,E2 2163} C_VEL
LIN {X 0,Y 578.531,Z 551.999,A -85,B 0,C 180,E1 2166.346,E2 2166.346} C_VEL
LIN {X 0,Y 578.628,Z 539.561,A -85,B 0,C 180,E1 2169.41,E2 2169.41} C_VEL
LIN {X 0,Y 578.844,Z 521.21,A -85,B 0,C 180,E1 2172.46,E2 2172.46} C_VEL
LIN {X 0,Y 579.251,Z 498.326,A -85,B 0,C 180,E1 2175.149,E2 2175.149} C_VEL
LIN {X 0,Y 579.743,Z 470.7,A -85,B 0,C 180,E1 2177.497,E2 2177.497} C_VEL
LIN {X 0,Y 580.323,Z 440.089,A -85,B 0,C 180,E1 2179.327,E2 2179.327} C_VEL
LIN {X 0,Y 580.778,Z 408.275,A -85,B 0,C 180,E1 2180.578,E2 2180.578} C_VEL
LIN {X 0,Y 579.78,Z 376.64,A -85,B 0,C 180,E1 2181.315,E2 2181.315} C_VEL
LIN {X 0,Y 577.998,Z 370.16,A -85,B 0,C 180,E1 2181.511,E2 2181.511} C_VEL
LIN {X 0,Y 577.937,Z 370.16,A -85,B 0,C 180,E1 2187.051,E2 2187.051} C_VEL
LIN {X 0,Y 577.921,Z 370.16,A -85,B 0,C 180,E1 2191.594,E2 2191.594} C_VEL
LIN {X 0,Y 578.059,Z 370.16,A -85,B 0,C 180,E1 2197.038,E2 2197.038} C_VEL
LIN {X 0,Y 577.84,Z 370.16,A -85,B 0,C 180,E1 2202.935,E2 2202.935} C_VEL
LIN {X 0,Y 577.971,Z 370.16,A -85,B 0,C 180,E1 2207.172,E2 2207.172} C_VEL
LIN {X 0,Y 577.948,Z 370.16,A -85,B 0,C 180,E1 2212.955,E2 2212.955} C_VEL
LIN {X 0,Y 577.903,Z 370.16,A -85,B 0,C 180,E1 2218.406,E2 2218.406} C_VEL
LIN {X 0,Y 578.001,Z 370.16,A -85,B 0,C 180,E1 2223.562,E2 2223.562} C_VEL
LIN {X 0,Y 578.145,Z 370.16,A -85,B 0,C 180,E1 2228.438,E2 2228.438} C_VEL
LIN {X 0,Y 580.765,Z 383.275,A -85,B 0,C 180,E1 2228.735,E2 2228.735} C_VEL
LIN {X 0,Y 580.649,Z 417.701,A -85,B 0,C 180,E1 2229.642,E2 2229.642} C_VEL
LIN {X 0,Y 580.144,Z 449.39,A -85,B 0,C 180,E1 2231.063,E2 2231.063} C_VEL
LIN {X 0,Y 579.599,Z 479.541,A -85,B 0,C 180,E1 2233.077,E2 2233.077} C_VEL
LIN {X 0,Y 579.157,Z 504.655,A -85,B 0,C 180,E1 2235.422,E2 2235.422} C_VEL
LIN {X 0,Y 578.857,Z 527.065,A -85,B 0,C 180,E1 2238.311,E2 2238.311} C_VEL
LIN {X 0,Y 578.639,Z 543.575,A -85,B 0,C 180,E1 2241.35,E2 2241.35} C_VEL
LIN {X 0,Y 578.553,Z 555.377,A -85,B 0,C 180,E1 2244.747,E2 2244.747} C_VEL
LIN {X 0,Y 578.416,Z 559.886,A -85,B 0,C 180,E1 2247.002,E2 2247.002} C_VEL
LIN {X 0,Y 578.418,Z 561.996,A -85,B 0,C 180,E1 2250.002,E2 2250.002} C_VEL
LIN {X 0,Y 578.443,Z 559.735,A -85,B 0,C 180,E1 2253.003,E2 2253.003} C_VEL
LIN {X 0,Y 578.536,Z 552.789,A -85,B 0,C 180,E1 2256.087,E2 2256.087} C_VEL
LIN {X 0,Y 578.631,Z 539.564,A -85,B 0,C 180,E1 2259.414,E2 2259.414} C_VEL
LIN {X 0,Y 578.846,Z 521.177,A -85,B 0,C 180,E1 2262.463,E2 2262.463} C_VEL
LIN {X 0,Y 579.266,Z 498.301,A -85,B 0,C 180,E1 2265.153,E2 2265.153} C_VEL
LIN {X 0,Y 579.784,Z 470.744,A -85,B 0,C 180,E1 2267.496,E2 2267.496} C_VEL
LIN {X 0,Y 580.341,Z 440.094,A -85,B 0,C 180,E1 2269.33,E2 2269.33} C_VEL
LIN {X 0,Y 580.813,Z 408.279,A -85,B 0,C 180,E1 2270.574,E2 2270.574} C_VEL
LIN {X 0,Y 579.854,Z 377.457,A -85,B 0,C 180,E1 2271.3,E2 2271.3} C_VEL
LIN {X 0,Y 577.959,Z 370.16,A -85,B 0,C 180,E1 2271.516,E2 2271.516} C_VEL
LIN {X 0,Y 577.92,Z 370.16,A -85,B 0,C 180,E1 2277.046,E2 2277.046} C_VEL
LIN {X 0,Y 577.982,Z 370.16,A -85,B 0,C 180,E1 2283.374,E2 2283.374} C_VEL
LIN {X 0,Y 577.835,Z 370.16,A -85,B 0,C 180,E1 2288.965,E2 2288.965} C_VEL
LIN {X 0,Y 577.912,Z 370.16,A -85,B 0,C 180,E1 2295.019,E2 2295.019} C_VEL
LIN {X 0,Y 577.86,Z 370.16,A -85,B 0,C 180,E1 2301.042,E2 2301.042} C_VEL
LIN {X 0,Y 577.785,Z 370.16,A -85,B 0,C 180,E1 2306.983,E2 2306.983} C_VEL
LIN {X 0,Y 577.874,Z 370.16,A -85,B 0,C 180,E1 2311.865,E2 2311.865} C_VEL
LIN {X 0,Y 577.946,Z 370.16,A -85,B 0,C 180,E1 2316.865,E2 2316.865} C_VEL
LIN {X 0,Y 578.096,Z 370.16,A -85,B 0,C 180,E1 2321.685,E2 2321.685} C_VEL
LIN {X 0,Y 578.287,Z 370.16,A -85,B 0,C 180,E1 2326.373,E2 2326.373} C_VEL
LIN {X 0,Y 578.175,Z 370.16,A -85,B 0,C 180,E1 2332.478,E2 2332.478} C_VEL
LIN {X 0,Y 578.311,Z 370.16,A -85,B 0,C 180,E1 2337,E2 2337} C_VEL
LIN {X 0,Y 578.379,Z 370.16,A -85,B 0,C 180,E1 2341.501,E2 2341.501} C_VEL
LIN {X 0,Y 578.372,Z 370.16,A -85,B 0,C 180,E1 2346.011,E2 2346.011} C_VEL
LIN {X 0,Y 578.045,Z 370.16,A -85,B 0,C 180,E1 2347.628,E2 2347.628} C_VEL
LIN {X 0,Y 574.153,Z 370.16,A -85,B 0,C 180,E1 2349.32,E2 2349.32} C_VEL
LIN {X 0,Y 570.214,Z 370.16,A -85,B 0,C 180,E1 2351.035,E2 2351.035} C_VEL
LIN {X 0,Y 570.075,Z 370.16,A -85,B 0,C 180,E1 2357.044,E2 2357.044} C_VEL
LIN {X 0,Y 570.11,Z 370.16,A -85,B 0,C 180,E1 2361.826,E2 2361.826} C_VEL
LIN {X 0,Y 570.029,Z 370.16,A -85,B 0,C 180,E1 2366.841,E2 2366.841} C_VEL
LIN {X 0,Y 569.921,Z 370.16,A -85,B 0,C 180,E1 2372.092,E2 2372.092} C_VEL
LIN {X 0,Y 570.127,Z 370.16,A -85,B 0,C 180,E1 2377.644,E2 2377.644} C_VEL
LIN {X 0,Y 569.917,Z 370.16,A -85,B 0,C 180,E1 2384.171,E2 2384.171} C_VEL
LIN {X 0,Y 569.956,Z 370.16,A -85,B 0,C 180,E1 2390.392,E2 2390.392} C_VEL
LIN {X 0,Y 569.874,Z 370.16,A -85,B 0,C 180,E1 2395.442,E2 2395.442} C_VEL
LIN {X 0,Y 569.956,Z 370.16,A -85,B 0,C 180,E1 2401.23,E2 2401.23} C_VEL
LIN {X 0,Y 570.096,Z 370.16,A -85,B 0,C 180,E1 2402.619,E2 2402.619} C_VEL
LIN {X 0,Y 575.012,Z 385.297,A -85,B 0,C 180,E1 2403.093,E2 2403.093} C_VEL
LIN {X 0,Y 574.736,Z 440.673,A -85,B 0,C 180,E1 2403.988,E2 2403.988} C_VEL
LIN {X 0,Y 574.145,Z 477.364,A -85,B 0,C 180,E1 2405.203,E2 2405.203} C_VEL
LIN {X 0,Y 573.316,Z 511.601,A -85,B 0,C 180,E1 2406.95,E2 2406.95} C_VEL
LIN {X 0,Y 572.443,Z 544.145,A -85,B 0,C 180,E1 2409.282,E2 2409.282} C_VEL
LIN {X 0,Y 571.701,Z 572.586,A -85,B 0,C 180,E1 2412.051,E2 2412.051} C_VEL
LIN {X 0,Y 571.106,Z 596.623,A -85,B 0,C 180,E1 2415.164,E2 2415.164} C_VEL
LIN {X 0,Y 570.806,Z 615.251,A -85,B 0,C 180,E1 2418.431,E2 2418.431} C_VEL
LIN {X 0,Y 570.634,Z 629.454,A -85,B 0,C 180,E1 2421.991,E2 2421.991} C_VEL
LIN {X 0,Y 570.542,Z 637.965,A -85,B 0,C 180,E1 2425.432,E2 2425.432} C_VEL
LIN {X 0,Y 570.526,Z 641.507,A -85,B 0,C 180,E1 2428.477,E2 2428.477} C_VEL
LIN {X 0,Y 570.598,Z 641.51,A -85,B 0,C 180,E1 2431.518,E2 2431.518} C_VEL
LIN {X 0,Y 570.582,Z 636.769,A -85,B 0,C 180,E1 2435.174,E2 2435.174} C_VEL
LIN {X 0,Y 570.663,Z 626.846,A -85,B 0,C 180,E1 2438.772,E2 2438.772} C_VEL
LIN {X 0,Y 570.865,Z 610.851,A -85,B 0,C 180,E1 2442.441,E2 2442.441} C_VEL
LIN {X 0,Y 571.249,Z 590.222,A -85,B 0,C 180,E1 2445.76,E2 2445.76} C_VEL
LIN {X 0,Y 571.876,Z 565.499,A -85,B 0,C 180,E1 2448.715,E2 2448.715} C_VEL
LIN {X 0,Y 572.685,Z 535.467,A -85,B 0,C 180,E1 2451.414,E2 2451.414} C_VEL
LIN {X 0,Y 573.639,Z 501.092,A -85,B 0,C 180,E1 2453.654,E2 2453.654} C_VEL
LIN {X 0,Y 574.36,Z 467.412,A -85,B 0,C 180,E1 2455.188,E2 2455.188} C_VEL
LIN {X 0,Y 574.895,Z 432.56,A -85,B 0,C 180,E1 2456.191,E2 2456.191} C_VEL
LIN {X 0,Y 574.43,Z 381.224,A -85,B 0,C 180,E1 2456.993,E2 2456.993} C_VEL
LIN {X 0,Y 570.34,Z 370.16,A -85,B 0,C 180,E1 2457.408,E2 2457.408} C_VEL
LIN {X 0,Y 570.119,Z 370.16,A -85,B 0,C 180,E1 2463.89,E2 2463.89} C_VEL
LIN {X 0,Y 569.95,Z 370.16,A -85,B 0,C 180,E1 2469.618,E2 2469.618} C_VEL
LIN {X 0,Y 569.779,Z 370.16,A -85,B 0,C 180,E1 2475.837,E2 2475.837} C_VEL
LIN {X 0,Y 569.811,Z 370.16,A -85,B 0,C 180,E1 2480.395,E2 2480.395} C_VEL
LIN {X 0,Y 569.88,Z 370.16,A -85,B 0,C 180,E1 2486.09,E2 2486.09} C_VEL
LIN {X 0,Y 569.967,Z 370.16,A -85,B 0,C 180,E1 2491.437,E2 2491.437} C_VEL
LIN {X 0,Y 570.11,Z 370.16,A -85,B 0,C 180,E1 2496.526,E2 2496.526} C_VEL
LIN {X 0,Y 570.188,Z 370.16,A -85,B 0,C 180,E1 2498.095,E2 2498.095} C_VEL
LIN {X 0,Y 573.475,Z 383.605,A -85,B 0,C 180,E1 2498.461,E2 2498.461} C_VEL
LIN {X 0,Y 573.235,Z 417.025,A -85,B 0,C 180,E1 2499.346,E2 2499.346} C_VEL
LIN {X 0,Y 572.693,Z 447.489,A -85,B 0,C 180,E1 2500.704,E2 2500.704} C_VEL
LIN {X 0,Y 572.004,Z 477.485,A -85,B 0,C 180,E1 2502.68,E2 2502.68} C_VEL
LIN {X 0,Y 571.418,Z 504.654,A -85,B 0,C 180,E1 2505.216,E2 2505.216} C_VEL
LIN {X 0,Y 571.017,Z 526.523,A -85,B 0,C 180,E1 2508.068,E2 2508.068} C_VEL
LIN {X 0,Y 570.749,Z 543.577,A -85,B 0,C 180,E1 2511.226,E2 2511.226} C_VEL
LIN {X 0,Y 570.674,Z 555.635,A -85,B 0,C 180,E1 2514.77,E2 2514.77} C_VEL
LIN {X 0,Y 570.526,Z 559.853,A -85,B 0,C 180,E1 2516.957,E2 2516.957} C_VEL
LIN {X 0,Y 570.539,Z 561.999,A -85,B 0,C 180,E1 2519.999,E2 2519.999} C_VEL
LIN {X 0,Y 570.523,Z 559.731,A -85,B 0,C 180,E1 2523.041,E2 2523.041} C_VEL
LIN {X 0,Y 570.627,Z 551.886,A -85,B 0,C 180,E1 2526.473,E2 2526.473} C_VEL
LIN {X 0,Y 570.768,Z 539.559,A -85,B 0,C 180,E1 2529.541,E2 2529.541} C_VEL
LIN {X 0,Y 571.047,Z 521.218,A -85,B 0,C 180,E1 2532.633,E2 2532.633} C_VEL
LIN {X 0,Y 571.551,Z 498.324,A -85,B 0,C 180,E1 2535.359,E2 2535.359} C_VEL
LIN {X 0,Y 572.142,Z 470.923,A -85,B 0,C 180,E1 2537.722,E2 2537.722} C_VEL
LIN {X 0,Y 572.812,Z 441.111,A -85,B 0,C 180,E1 2539.541,E2 2539.541} C_VEL
LIN {X 0,Y 573.374,Z 408.617,A -85,B 0,C 180,E1 2540.847,E2 2540.847} C_VEL
LIN {X 0,Y 572.644,Z 379.182,A -85,B 0,C 180,E1 2541.554,E2 2541.554} C_VEL
LIN {X 0,Y 570.068,Z 370.16,A -85,B 0,C 180,E1 2541.825,E2 2541.825} C_VEL
LIN {X 0,Y 570.085,Z 370.16,A -85,B 0,C 180,E1 2546.836,E2 2546.836} C_VEL
LIN {X 0,Y 569.988,Z 370.16,A -85,B 0,C 180,E1 2552.086,E2 2552.086} C_VEL
LIN {X 0,Y 570.143,Z 370.16,A -85,B 0,C 180,E1 2557.64,E2 2557.64} C_VEL
LIN {X 0,Y 569.898,Z 370.16,A -85,B 0,C 180,E1 2564.175,E2 2564.175} C_VEL
LIN {X 0,Y 569.983,Z 370.16,A -85,B 0,C 180,E1 2568.396,E2 2568.396} C_VEL
LIN {X 0,Y 570.001,Z 370.16,A -85,B 0,C 180,E1 2574.248,E2 2574.248} C_VEL
LIN {X 0,Y 570.023,Z 370.16,A -85,B 0,C 180,E1 2579.696,E2 2579.696} C_VEL
LIN {X 0,Y 570.125,Z 370.16,A -85,B 0,C 180,E1 2584.86,E2 2584.86} C_VEL
LIN {X 0,Y 570.203,Z 370.16,A -85,B 0,C 180,E1 2588.112,E2 2588.112} C_VEL
LIN {X 0,Y 573.418,Z 384.062,A -85,B 0,C 180,E1 2588.462,E2 2588.462} C_VEL
LIN {X 0,Y 573.205,Z 418.72,A -85,B 0,C 180,E1 2589.403,E2 2589.403} C_VEL
LIN {X 0,Y 572.566,Z 451.079,A -85,B 0,C 180,E1 2590.903,E2 2590.903} C_VEL
LIN {X 0,Y 571.91,Z 481.156,A -85,B 0,C 180,E1 2592.973,E2 2592.973} C_VEL
LIN {X 0,Y 571.371,Z 506.858,A -85,B 0,C 180,E1 2595.466,E2 2595.466} C_VEL
LIN {X 0,Y 571.01,Z 528.537,A -85,B 0,C 180,E1 2598.384,E2 2598.384} C_VEL
LIN {X 0,Y 570.746,Z 545.217,A -85,B 0,C 180,E1 2601.613,E2 2601.613} C_VEL
LIN {X 0,Y 570.668,Z 555.644,A -85,B 0,C 180,E1 2604.781,E2 2604.781} C_VEL
LIN {X 0,Y 570.519,Z 559.886,A -85,B 0,C 180,E1 2606.96,E2 2606.96} C_VEL
LIN {X 0,Y 570.548,Z 561.996,A -85,B 0,C 180,E1 2610.002,E2 2610.002} C_VEL
LIN {X 0,Y 570.544,Z 559.737,A -85,B 0,C 180,E1 2613.044,E2 2613.044} C_VEL
LIN {X 0,Y 570.627,Z 551.876,A -85,B 0,C 180,E1 2616.477,E2 2616.477} C_VEL
LIN {X 0,Y 570.771,Z 539.567,A -85,B 0,C 180,E1 2619.545,E2 2619.545} C_VEL
LIN {X 0,Y 571.041,Z 521.183,A -85,B 0,C 180,E1 2622.636,E2 2622.636} C_VEL
LIN {X 0,Y 571.56,Z 498.306,A -85,B 0,C 180,E1 2625.362,E2 2625.362} C_VEL
LIN {X 0,Y 572.144,Z 470.98,A -85,B 0,C 180,E1 2627.721,E2 2627.721} C_VEL
LIN {X 0,Y 572.833,Z 440.103,A -85,B 0,C 180,E1 2629.594,E2 2629.594} C_VEL
LIN {X 0,Y 573.408,Z 408.474,A -85,B 0,C 180,E1 2630.847,E2 2630.847} C_VEL
LIN {X 0,Y 572.648,Z 379.556,A -85,B 0,C 180,E1 2631.549,E2 2631.549} C_VEL
LIN {X 0,Y 570.062,Z 370.16,A -85,B 0,C 180,E1 2631.829,E2 2631.829} C_VEL
LIN {X 0,Y 570.026,Z 370.16,A -85,B 0,C 180,E1 2636.843,E2 2636.843} C_VEL
LIN {X 0,Y 569.974,Z 370.16,A -85,B 0,C 180,E1 2642.091,E2 2642.091} C_VEL
LIN {X 0,Y 569.864,Z 370.16,A -85,B 0,C 180,E1 2647.667,E2 2647.667} C_VEL
LIN {X 0,Y 569.866,Z 370.16,A -85,B 0,C 180,E1 2653.691,E2 2653.691} C_VEL
LIN {X 0,Y 569.951,Z 370.16,A -85,B 0,C 180,E1 2658.392,E2 2658.392} C_VEL
LIN {X 0,Y 569.918,Z 370.16,A -85,B 0,C 180,E1 2664.241,E2 2664.241} C_VEL
LIN {X 0,Y 569.977,Z 370.16,A -85,B 0,C 180,E1 2669.693,E2 2669.693} C_VEL
LIN {X 0,Y 570.131,Z 370.16,A -85,B 0,C 180,E1 2674.859,E2 2674.859} C_VEL
LIN {X 0,Y 570.191,Z 370.16,A -85,B 0,C 180,E1 2679.809,E2 2679.809} C_VEL
LIN {X 0,Y 570.363,Z 370.16,A -85,B 0,C 180,E1 2686.18,E2 2686.18} C_VEL
LIN {X 0,Y 570.266,Z 370.16,A -85,B 0,C 180,E1 2692.373,E2 2692.373} C_VEL
LIN {X 0,Y 570.403,Z 370.16,A -85,B 0,C 180,E1 2696.958,E2 2696.958} C_VEL
LIN {X 0,Y 570.482,Z 370.16,A -85,B 0,C 180,E1 2701.522,E2 2701.522} C_VEL
LIN {X 0,Y 570.441,Z 370.16,A -85,B 0,C 180,E1 2706.095,E2 2706.095} C_VEL
LIN {X 0,Y 570.214,Z 370.16,A -85,B 0,C 180,E1 2711.035,E2 2711.035} C_VEL
LIN {X 0,Y 566.159,Z 370.16,A -85,B 0,C 180,E1 2712.747,E2 2712.747} C_VEL
LIN {X 0,Y 562.184,Z 370.16,A -85,B 0,C 180,E1 2714.482,E2 2714.482} C_VEL
LIN {X 0,Y 562.237,Z 370.16,A -85,B 0,C 180,E1 2720.491,E2 2720.491} C_VEL
LIN {X 0,Y 562.205,Z 370.16,A -85,B 0,C 180,E1 2725.523,E2 2725.523} C_VEL
LIN {X 0,Y 562.041,Z 370.16,A -85,B 0,C 180,E1 2730.784,E2 2730.784} C_VEL
LIN {X 0,Y 562.147,Z 370.16,A -85,B 0,C 180,E1 2736.334,E2 2736.334} C_VEL
LIN {X 0,Y 561.95,Z 370.16,A -85,B 0,C 180,E1 2742.34,E2 2742.34} C_VEL
LIN {X 0,Y 562.019,Z 370.16,A -85,B 0,C 180,E1 2747.664,E2 2747.664} C_VEL
LIN {X 0,Y 562.086,Z 370.16,A -85,B 0,C 180,E1 2753.904,E2 2753.904} C_VEL
LIN {X 0,Y 562.062,Z 370.16,A -85,B 0,C 180,E1 2759.534,E2 2759.534} C_VEL
LIN {X 0,Y 562.111,Z 370.16,A -85,B 0,C 180,E1 2762.206,E2 2762.206} C_VEL
LIN {X 0,Y 568.001,Z 387.506,A -85,B 0,C 180,E1 2762.764,E2 2762.764} C_VEL
LIN {X 0,Y 567.619,Z 441.405,A -85,B 0,C 180,E1 2763.656,E2 2763.656} C_VEL
LIN {X 0,Y 566.903,Z 478.231,A -85,B 0,C 180,E1 2764.902,E2 2764.902} C_VEL
LIN {X 0,Y 565.906,Z 512.782,A -85,B 0,C 180,E1 2766.703,E2 2766.703} C_VEL
LIN {X 0,Y 564.881,Z 545.294,A -85,B 0,C 180,E1 2769.095,E2 2769.095} C_VEL
LIN {X 0,Y 563.993,Z 574.103,A -85,B 0,C 180,E1 2771.972,E2 2771.972} C_VEL
LIN {X 0,Y 563.317,Z 598.5,A -85,B 0,C 180,E1 2775.241,E2 2775.241} C_VEL
LIN {X 0,Y 562.882,Z 617.675,A -85,B 0,C 180,E1 2778.799,E2 2778.799} C_VEL
LIN {X 0,Y 562.73,Z 630.601,A -85,B 0,C 180,E1 2782.267,E2 2782.267} C_VEL
LIN {X 0,Y 562.65,Z 637.964,A -85,B 0,C 180,E1 2785.368,E2 2785.368} C_VEL
LIN {X 0,Y 562.624,Z 641.507,A -85,B 0,C 180,E1 2788.456,E2 2788.456} C_VEL
LIN {X 0,Y 562.694,Z 641.51,A -85,B 0,C 180,E1 2791.539,E2 2791.539} C_VEL
LIN {X 0,Y 562.659,Z 636.447,A -85,B 0,C 180,E1 2795.408,E2 2795.408} C_VEL
LIN {X 0,Y 562.776,Z 626.846,A -85,B 0,C 180,E1 2798.896,E2 2798.896} C_VEL
LIN {X 0,Y 563.007,Z 610.852,A -85,B 0,C 180,E1 2802.618,E2 2802.618} C_VEL
LIN {X 0,Y 563.482,Z 590.221,A -85,B 0,C 180,E1 2805.983,E2 2805.983} C_VEL
LIN {X 0,Y 564.242,Z 563.978,A -85,B 0,C 180,E1 2809.14,E2 2809.14} C_VEL
LIN {X 0,Y 565.248,Z 534.188,A -85,B 0,C 180,E1 2811.813,E2 2811.813} C_VEL
LIN {X 0,Y 566.331,Z 499.893,A -85,B 0,C 180,E1 2814.045,E2 2814.045} C_VEL
LIN {X 0,Y 567.255,Z 465.507,A -85,B 0,C 180,E1 2815.599,E2 2815.599} C_VEL
LIN {X 0,Y 567.926,Z 428.698,A -85,B 0,C 180,E1 2816.622,E2 2816.622} C_VEL
LIN {X 0,Y 567.24,Z 383.019,A -85,B 0,C 180,E1 2817.338,E2 2817.338} C_VEL
LIN {X 0,Y 562.367,Z 370.16,A -85,B 0,C 180,E1 2817.819,E2 2817.819} C_VEL
LIN {X 0,Y 562.225,Z 370.16,A -85,B 0,C 180,E1 2824.433,E2 2824.433} C_VEL
LIN {X 0,Y 561.983,Z 370.16,A -85,B 0,C 180,E1 2830.278,E2 2830.278} C_VEL
LIN {X 0,Y 561.843,Z 370.16,A -85,B 0,C 180,E1 2835.525,E2 2835.525} C_VEL
LIN {X 0,Y 561.869,Z 370.16,A -85,B 0,C 180,E1 2841.384,E2 2841.384} C_VEL
LIN {X 0,Y 561.947,Z 370.16,A -85,B 0,C 180,E1 2846.629,E2 2846.629} C_VEL
LIN {X 0,Y 562.08,Z 370.16,A -85,B 0,C 180,E1 2850.999,E2 2850.999} C_VEL
LIN {X 0,Y 562.184,Z 370.16,A -85,B 0,C 180,E1 2856.285,E2 2856.285} C_VEL
LIN {X 0,Y 562.276,Z 370.16,A -85,B 0,C 180,E1 2857.806,E2 2857.806} C_VEL
LIN {X 0,Y 566.117,Z 385.002,A -85,B 0,C 180,E1 2858.192,E2 2858.192} C_VEL
LIN {X 0,Y 565.765,Z 420.365,A -85,B 0,C 180,E1 2859.183,E2 2859.183} C_VEL
LIN {X 0,Y 565.034,Z 452.717,A -85,B 0,C 180,E1 2860.737,E2 2860.737} C_VEL
LIN {X 0,Y 564.245,Z 482.217,A -85,B 0,C 180,E1 2862.833,E2 2862.833} C_VEL
LIN {X 0,Y 563.596,Z 507.93,A -85,B 0,C 180,E1 2865.389,E2 2865.389} C_VEL
LIN {X 0,Y 563.152,Z 529.611,A -85,B 0,C 180,E1 2868.392,E2 2868.392} C_VEL
LIN {X 0,Y 562.879,Z 545.173,A -85,B 0,C 180,E1 2871.492,E2 2871.492} C_VEL
LIN {X 0,Y 562.774,Z 555.71,A -85,B 0,C 180,E1 2874.725,E2 2874.725} C_VEL
LIN {X 0,Y 562.629,Z 559.847,A -85,B 0,C 180,E1 2876.914,E2 2876.914} C_VEL
LIN {X 0,Y 562.64,Z 561.999,A -85,B 0,C 180,E1 2879.999,E2 2879.999} C_VEL
LIN {X 0,Y 562.624,Z 559.731,A -85,B 0,C 180,E1 2883.084,E2 2883.084} C_VEL
LIN {X 0,Y 562.742,Z 551.888,A -85,B 0,C 180,E1 2886.564,E2 2886.564} C_VEL
LIN {X 0,Y 562.913,Z 539.556,A -85,B 0,C 180,E1 2889.676,E2 2889.676} C_VEL
LIN {X 0,Y 563.223,Z 521.226,A -85,B 0,C 180,E1 2892.811,E2 2892.811} C_VEL
LIN {X 0,Y 563.825,Z 498.32,A -85,B 0,C 180,E1 2895.574,E2 2895.574} C_VEL
LIN {X 0,Y 564.491,Z 472.207,A -85,B 0,C 180,E1 2897.876,E2 2897.876} C_VEL
LIN {X 0,Y 565.308,Z 442.132,A -85,B 0,C 180,E1 2899.76,E2 2899.76} C_VEL
LIN {X 0,Y 565.975,Z 408.648,A -85,B 0,C 180,E1 2901.132,E2 2901.132} C_VEL
LIN {X 0,Y 565.082,Z 380.043,A -85,B 0,C 180,E1 2901.843,E2 2901.843} C_VEL
LIN {X 0,Y 562.137,Z 370.16,A -85,B 0,C 180,E1 2902.149,E2 2902.149} C_VEL
LIN {X 0,Y 562.121,Z 370.16,A -85,B 0,C 180,E1 2907.286,E2 2907.286} C_VEL
LIN {X 0,Y 562.013,Z 370.16,A -85,B 0,C 180,E1 2912.597,E2 2912.597} C_VEL
LIN {X 0,Y 562.137,Z 370.16,A -85,B 0,C 180,E1 2918.272,E2 2918.272} C_VEL
LIN {X 0,Y 562.006,Z 370.16,A -85,B 0,C 180,E1 2924.456,E2 2924.456} C_VEL
LIN {X 0,Y 562.026,Z 370.16,A -85,B 0,C 180,E1 2929.726,E2 2929.726} C_VEL
LIN {X 0,Y 561.998,Z 370.16,A -85,B 0,C 180,E1 2935.552,E2 2935.552} C_VEL
LIN {X 0,Y 562.072,Z 370.16,A -85,B 0,C 180,E1 2941.002,E2 2941.002} C_VEL
LIN {X 0,Y 562.181,Z 370.16,A -85,B 0,C 180,E1 2946.287,E2 2946.287} C_VEL
LIN {X 0,Y 562.268,Z 370.16,A -85,B 0,C 180,E1 2947.76,E2 2947.76} C_VEL
LIN {X 0,Y 566.081,Z 383.94,A -85,B 0,C 180,E1 2948.168,E2 2948.168} C_VEL
LIN {X 0,Y 565.795,Z 418.387,A -85,B 0,C 180,E1 2949.11,E2 2949.11} C_VEL
LIN {X 0,Y 565.04,Z 451.064,A -85,B 0,C 180,E1 2950.639,E2 2950.639} C_VEL
LIN {X 0,Y 564.278,Z 480.494,A -85,B 0,C 180,E1 2952.68,E2 2952.68} C_VEL
LIN {X 0,Y 563.604,Z 506.631,A -85,B 0,C 180,E1 2955.236,E2 2955.236} C_VEL
LIN {X 0,Y 563.162,Z 527.948,A -85,B 0,C 180,E1 2958.125,E2 2958.125} C_VEL
LIN {X 0,Y 562.882,Z 543.568,A -85,B 0,C 180,E1 2961.106,E2 2961.106} C_VEL
LIN {X 0,Y 562.727,Z 555.123,A -85,B 0,C 180,E1 2964.498,E2 2964.498} C_VEL
LIN {X 0,Y 562.622,Z 559.886,A -85,B 0,C 180,E1 2966.917,E2 2966.917} C_VEL
LIN {X 0,Y 562.649,Z 561.996,A -85,B 0,C 180,E1 2970.002,E2 2970.002} C_VEL
LIN {X 0,Y 562.646,Z 559.739,A -85,B 0,C 180,E1 2973.087,E2 2973.087} C_VEL
LIN {X 0,Y 562.747,Z 551.878,A -85,B 0,C 180,E1 2976.568,E2 2976.568} C_VEL
LIN {X 0,Y 562.916,Z 539.569,A -85,B 0,C 180,E1 2979.679,E2 2979.679} C_VEL
LIN {X 0,Y 563.216,Z 521.189,A -85,B 0,C 180,E1 2982.815,E2 2982.815} C_VEL
LIN {X 0,Y 563.834,Z 498.311,A -85,B 0,C 180,E1 2985.578,E2 2985.578} C_VEL
LIN {X 0,Y 564.546,Z 470.992,A -85,B 0,C 180,E1 2987.968,E2 2987.968} C_VEL
LIN {X 0,Y 565.349,Z 440.113,A -85,B 0,C 180,E1 2989.864,E2 2989.864} C_VEL
LIN {X 0,Y 566.008,Z 407.319,A -85,B 0,C 180,E1 2991.169,E2 2991.169} C_VEL
LIN {X 0,Y 565.058,Z 380.385,A -85,B 0,C 180,E1 2991.841,E2 2991.841} C_VEL
LIN {X 0,Y 562.139,Z 370.16,A -85,B 0,C 180,E1 2992.153,E2 2992.153} C_VEL
LIN {X 0,Y 562.074,Z 370.16,A -85,B 0,C 180,E1 2997.275,E2 2997.275} C_VEL
LIN {X 0,Y 562.043,Z 370.16,A -85,B 0,C 180,E1 3003.385,E2 3003.385} C_VEL
LIN {X 0,Y 561.896,Z 370.16,A -85,B 0,C 180,E1 3008.618,E2 3008.618} C_VEL
LIN {X 0,Y 561.975,Z 370.16,A -85,B 0,C 180,E1 3014.464,E2 3014.464} C_VEL
LIN {X 0,Y 562,Z 370.16,A -85,B 0,C 180,E1 3019.723,E2 3019.723} C_VEL
LIN {X 0,Y 561.932,Z 370.16,A -85,B 0,C 180,E1 3025.546,E2 3025.546} C_VEL
LIN {X 0,Y 562.019,Z 370.16,A -85,B 0,C 180,E1 3030.998,E2 3030.998} C_VEL
LIN {X 0,Y 562.191,Z 370.16,A -85,B 0,C 180,E1 3036.295,E2 3036.295} C_VEL
LIN {X 0,Y 562.264,Z 370.16,A -85,B 0,C 180,E1 3041.15,E2 3041.15} C_VEL
LIN {X 0,Y 562.419,Z 370.16,A -85,B 0,C 180,E1 3045.981,E2 3045.981} C_VEL
LIN {X 0,Y 562.359,Z 370.16,A -85,B 0,C 180,E1 3052.265,E2 3052.265} C_VEL
LIN {X 0,Y 562.495,Z 370.16,A -85,B 0,C 180,E1 3056.915,E2 3056.915} C_VEL
LIN {X 0,Y 562.571,Z 370.16,A -85,B 0,C 180,E1 3061.543,E2 3061.543} C_VEL
LIN {X 0,Y 562.521,Z 370.16,A -85,B 0,C 180,E1 3066.181,E2 3066.181} C_VEL
LIN {X 0,Y 562.223,Z 370.16,A -85,B 0,C 180,E1 3072.441,E2 3072.441} C_VEL
LIN {X 0,Y 562.184,Z 370.16,A -85,B 0,C 180,E1 3074.482,E2 3074.482} C_VEL
LIN {X 0,Y 558.202,Z 370.16,A -85,B 0,C 180,E1 3076.225,E2 3076.225} C_VEL
LIN {X 0,Y 554.211,Z 370.16,A -85,B 0,C 180,E1 3077.992,E2 3077.992} C_VEL
LIN {X 0,Y 554.244,Z 370.16,A -85,B 0,C 180,E1 3082.484,E2 3082.484} C_VEL
LIN {X 0,Y 554.129,Z 370.16,A -85,B 0,C 180,E1 3087.676,E2 3087.676} C_VEL
LIN {X 0,Y 554.049,Z 370.16,A -85,B 0,C 180,E1 3093.128,E2 3093.128} C_VEL
LIN {X 0,Y 554.169,Z 370.16,A -85,B 0,C 180,E1 3098.928,E2 3098.928} C_VEL
LIN {X 0,Y 554.135,Z 370.16,A -85,B 0,C 180,E1 3105.263,E2 3105.263} C_VEL
LIN {X 0,Y 554.11,Z 370.16,A -85,B 0,C 180,E1 3111.065,E2 3111.065} C_VEL
LIN {X 0,Y 554.031,Z 370.16,A -85,B 0,C 180,E1 3116.869,E2 3116.869} C_VEL
LIN {X 0,Y 554.211,Z 370.249,A -85,B 0,C 180,E1 3121.779,E2 3121.779} C_VEL
LIN {X 0,Y 561.04,Z 390.201,A -85,B 0,C 180,E1 3122.436,E2 3122.436} C_VEL
LIN {X 0,Y 560.52,Z 442.042,A -85,B 0,C 180,E1 3123.314,E2 3123.314} C_VEL
LIN {X 0,Y 559.667,Z 478.607,A -85,B 0,C 180,E1 3124.572,E2 3124.572} C_VEL
LIN {X 0,Y 558.51,Z 514.208,A -85,B 0,C 180,E1 3126.466,E2 3126.466} C_VEL
LIN {X 0,Y 557.315,Z 546.443,A -85,B 0,C 180,E1 3128.901,E2 3128.901} C_VEL
LIN {X 0,Y 556.301,Z 574.185,A -85,B 0,C 180,E1 3131.724,E2 3131.724} C_VEL
LIN {X 0,Y 555.562,Z 597.805,A -85,B 0,C 180,E1 3134.92,E2 3134.92} C_VEL
LIN {X 0,Y 555.057,Z 617.474,A -85,B 0,C 180,E1 3138.592,E2 3138.592} C_VEL
LIN {X 0,Y 554.843,Z 630.601,A -85,B 0,C 180,E1 3142.156,E2 3142.156} C_VEL
LIN {X 0,Y 554.762,Z 637.964,A -85,B 0,C 180,E1 3145.302,E2 3145.302} C_VEL
LIN {X 0,Y 554.722,Z 641.507,A -85,B 0,C 180,E1 3148.434,E2 3148.434} C_VEL
LIN {X 0,Y 554.789,Z 641.511,A -85,B 0,C 180,E1 3151.561,E2 3151.561} C_VEL
LIN {X 0,Y 554.756,Z 636.447,A -85,B 0,C 180,E1 3155.485,E2 3155.485} C_VEL
LIN {X 0,Y 554.886,Z 626.846,A -85,B 0,C 180,E1 3159.024,E2 3159.024} C_VEL
LIN {X 0,Y 555.186,Z 610.853,A -85,B 0,C 180,E1 3162.798,E2 3162.798} C_VEL
LIN {X 0,Y 555.71,Z 590.219,A -85,B 0,C 180,E1 3166.213,E2 3166.213} C_VEL
LIN {X 0,Y 556.606,Z 564.382,A -85,B 0,C 180,E1 3169.369,E2 3169.369} C_VEL
LIN {X 0,Y 557.805,Z 534.188,A -85,B 0,C 180,E1 3172.119,E2 3172.119} C_VEL
LIN {X 0,Y 558.999,Z 501.359,A -85,B 0,C 180,E1 3174.298,E2 3174.298} C_VEL
LIN {X 0,Y 560.039,Z 466.923,A -85,B 0,C 180,E1 3175.898,E2 3175.898} C_VEL
LIN {X 0,Y 560.782,Z 431.85,A -85,B 0,C 180,E1 3176.918,E2 3176.918} C_VEL
LIN {X 0,Y 560.196,Z 385.119,A -85,B 0,C 180,E1 3177.682,E2 3177.682} C_VEL
LIN {X 0,Y 554.398,Z 370.16,A -85,B 0,C 180,E1 3178.28,E2 3178.28} C_VEL
LIN {X 0,Y 554.262,Z 370.16,A -85,B 0,C 180,E1 3184.999,E2 3184.999} C_VEL
LIN {X 0,Y 554.056,Z 370.16,A -85,B 0,C 180,E1 3190.976,E2 3190.976} C_VEL
LIN {X 0,Y 554.015,Z 370.16,A -85,B 0,C 180,E1 3197.542,E2 3197.542} C_VEL
LIN {X 0,Y 554.011,Z 370.16,A -85,B 0,C 180,E1 3203.044,E2 3203.044} C_VEL
LIN {X 0,Y 554.102,Z 370.16,A -85,B 0,C 180,E1 3208.726,E2 3208.726} C_VEL
LIN {X 0,Y 554.319,Z 370.16,A -85,B 0,C 180,E1 3214.321,E2 3214.321} C_VEL
LIN {X 0,Y 554.372,Z 370.16,A -85,B 0,C 180,E1 3217.521,E2 3217.521} C_VEL
LIN {X 0,Y 558.705,Z 385.715,A -85,B 0,C 180,E1 3217.93,E2 3217.93} C_VEL
LIN {X 0,Y 558.338,Z 419.887,A -85,B 0,C 180,E1 3218.882,E2 3218.882} C_VEL
LIN {X 0,Y 557.59,Z 450.149,A -85,B 0,C 180,E1 3220.32,E2 3220.32} C_VEL
LIN {X 0,Y 556.692,Z 478.56,A -85,B 0,C 180,E1 3222.282,E2 3222.282} C_VEL
LIN {X 0,Y 555.92,Z 504.843,A -85,B 0,C 180,E1 3224.816,E2 3224.816} C_VEL
LIN {X 0,Y 555.321,Z 526.974,A -85,B 0,C 180,E1 3227.802,E2 3227.802} C_VEL
LIN {X 0,Y 554.997,Z 543.555,A -85,B 0,C 180,E1 3230.975,E2 3230.975} C_VEL
LIN {X 0,Y 554.841,Z 555.094,A -85,B 0,C 180,E1 3234.397,E2 3234.397} C_VEL
LIN {X 0,Y 554.744,Z 559.841,A -85,B 0,C 180,E1 3236.87,E2 3236.87} C_VEL
LIN {X 0,Y 554.77,Z 561.999,A -85,B 0,C 180,E1 3239.999,E2 3239.999} C_VEL
LIN {X 0,Y 554.738,Z 559.73,A -85,B 0,C 180,E1 3243.128,E2 3243.128} C_VEL
LIN {X 0,Y 554.85,Z 551.89,A -85,B 0,C 180,E1 3246.658,E2 3246.658} C_VEL
LIN {X 0,Y 555.038,Z 539.553,A -85,B 0,C 180,E1 3249.814,E2 3249.814} C_VEL
LIN {X 0,Y 555.429,Z 521.233,A -85,B 0,C 180,E1 3252.994,E2 3252.994} C_VEL
LIN {X 0,Y 556.102,Z 498.317,A -85,B 0,C 180,E1 3255.796,E2 3255.796} C_VEL
LIN {X 0,Y 556.894,Z 472.497,A -85,B 0,C 180,E1 3258.107,E2 3258.107} C_VEL
LIN {X 0,Y 557.833,Z 441.572,A -85,B 0,C 180,E1 3260.064,E2 3260.064} C_VEL
LIN {X 0,Y 558.574,Z 409.152,A -85,B 0,C 180,E1 3261.402,E2 3261.402} C_VEL
LIN {X 0,Y 557.663,Z 381.843,A -85,B 0,C 180,E1 3262.095,E2 3262.095} C_VEL
LIN {X 0,Y 554.219,Z 370.16,A -85,B 0,C 180,E1 3262.483,E2 3262.483} C_VEL
LIN {X 0,Y 554.193,Z 370.16,A -85,B 0,C 180,E1 3267.67,E2 3267.67} C_VEL
LIN {X 0,Y 554.115,Z 370.16,A -85,B 0,C 180,E1 3273.121,E2 3273.121} C_VEL
LIN {X 0,Y 554.187,Z 370.16,A -85,B 0,C 180,E1 3278.924,E2 3278.924} C_VEL
LIN {X 0,Y 554.13,Z 370.16,A -85,B 0,C 180,E1 3285.26,E2 3285.26} C_VEL
LIN {X 0,Y 554.116,Z 370.16,A -85,B 0,C 180,E1 3291.071,E2 3291.071} C_VEL
LIN {X 0,Y 554.054,Z 370.16,A -85,B 0,C 180,E1 3296.876,E2 3296.876} C_VEL
LIN {X 0,Y 554.172,Z 370.16,A -85,B 0,C 180,E1 3302.33,E2 3302.33} C_VEL
LIN {X 0,Y 554.368,Z 370.16,A -85,B 0,C 180,E1 3307.351,E2 3307.351} C_VEL
LIN {X 0,Y 558.963,Z 385.999,A -85,B 0,C 180,E1 3307.858,E2 3307.858} C_VEL
LIN {X 0,Y 558.478,Z 418.987,A -85,B 0,C 180,E1 3308.811,E2 3308.811} C_VEL
LIN {X 0,Y 557.497,Z 451.77,A -85,B 0,C 180,E1 3310.41,E2 3310.41} C_VEL
LIN {X 0,Y 556.628,Z 480.551,A -85,B 0,C 180,E1 3312.44,E2 3312.44} C_VEL
LIN {X 0,Y 555.865,Z 506.625,A -85,B 0,C 180,E1 3315.026,E2 3315.026} C_VEL
LIN {X 0,Y 555.327,Z 528.244,A -85,B 0,C 180,E1 3318.005,E2 3318.005} C_VEL
LIN {X 0,Y 555.002,Z 543.564,A -85,B 0,C 180,E1 3320.978,E2 3320.978} C_VEL
LIN {X 0,Y 554.826,Z 555.121,A -85,B 0,C 180,E1 3324.42,E2 3324.42} C_VEL
LIN {X 0,Y 554.738,Z 559.886,A -85,B 0,C 180,E1 3326.873,E2 3326.873} C_VEL
LIN {X 0,Y 554.779,Z 561.997,A -85,B 0,C 180,E1 3330.002,E2 3330.002} C_VEL
LIN {X 0,Y 554.759,Z 559.741,A -85,B 0,C 180,E1 3333.131,E2 3333.131} C_VEL
LIN {X 0,Y 554.856,Z 551.88,A -85,B 0,C 180,E1 3336.661,E2 3336.661} C_VEL
LIN {X 0,Y 555.042,Z 539.572,A -85,B 0,C 180,E1 3339.818,E2 3339.818} C_VEL
LIN {X 0,Y 555.431,Z 521.195,A -85,B 0,C 180,E1 3342.998,E2 3342.998} C_VEL
LIN {X 0,Y 556.098,Z 498.316,A -85,B 0,C 180,E1 3345.8,E2 3345.8} C_VEL
LIN {X 0,Y 556.98,Z 471.201,A -85,B 0,C 180,E1 3348.205,E2 3348.205} C_VEL
LIN {X 0,Y 557.875,Z 439.96,A -85,B 0,C 180,E1 3350.158,E2 3350.158} C_VEL
LIN {X 0,Y 558.77,Z 408.081,A -85,B 0,C 180,E1 3351.478,E2 3351.478} C_VEL
LIN {X 0,Y 558.255,Z 383.043,A -85,B 0,C 180,E1 3352.144,E2 3352.144} C_VEL
LIN {X 0,Y 554.213,Z 370.16,A -85,B 0,C 180,E1 3352.582,E2 3352.582} C_VEL
LIN {X 0,Y 554.147,Z 370.16,A -85,B 0,C 180,E1 3357.677,E2 3357.677} C_VEL
LIN {X 0,Y 554.133,Z 370.16,A -85,B 0,C 180,E1 3363.124,E2 3363.124} C_VEL
LIN {X 0,Y 553.974,Z 370.16,A -85,B 0,C 180,E1 3368.947,E2 3368.947} C_VEL
LIN {X 0,Y 554.117,Z 370.16,A -85,B 0,C 180,E1 3375.267,E2 3375.267} C_VEL
LIN {X 0,Y 554.068,Z 370.16,A -85,B 0,C 180,E1 3381.066,E2 3381.066} C_VEL
LIN {X 0,Y 554.007,Z 370.16,A -85,B 0,C 180,E1 3386.872,E2 3386.872} C_VEL
LIN {X 0,Y 554.157,Z 370.16,A -85,B 0,C 180,E1 3392.328,E2 3392.328} C_VEL
LIN {X 0,Y 554.243,Z 370.16,A -85,B 0,C 180,E1 3397.518,E2 3397.518} C_VEL
LIN {X 0,Y 554.366,Z 370.16,A -85,B 0,C 180,E1 3402.914,E2 3402.914} C_VEL
LIN {X 0,Y 554.43,Z 370.16,A -85,B 0,C 180,E1 3407.383,E2 3407.383} C_VEL
LIN {X 0,Y 554.447,Z 370.16,A -85,B 0,C 180,E1 3412.154,E2 3412.154} C_VEL
LIN {X 0,Y 554.607,Z 370.16,A -85,B 0,C 180,E1 3416.871,E2 3416.871} C_VEL
LIN {X 0,Y 554.661,Z 370.16,A -85,B 0,C 180,E1 3421.565,E2 3421.565} C_VEL
LIN {X 0,Y 554.591,Z 370.16,A -85,B 0,C 180,E1 3426.27,E2 3426.27} C_VEL
LIN {X 0,Y 554.301,Z 370.16,A -85,B 0,C 180,E1 3432.622,E2 3432.622} C_VEL
LIN {X 0,Y 554.211,Z 370.16,A -85,B 0,C 180,E1 3437.992,E2 3437.992} C_VEL
LIN {X 0,Y 550.304,Z 370.16,A -85,B 0,C 180,E1 3439.758,E2 3439.758} C_VEL
LIN {X 0,Y 546.32,Z 370.16,A -85,B 0,C 180,E1 3441.548,E2 3441.548} C_VEL
LIN {X 0,Y 546.28,Z 370.16,A -85,B 0,C 180,E1 3446.323,E2 3446.323} C_VEL
LIN {X 0,Y 546.139,Z 370.16,A -85,B 0,C 180,E1 3451.783,E2 3451.783} C_VEL
LIN {X 0,Y 546.266,Z 370.16,A -85,B 0,C 180,E1 3457.569,E2 3457.569} C_VEL
LIN {X 0,Y 546.134,Z 370.16,A -85,B 0,C 180,E1 3463.881,E2 3463.881} C_VEL
LIN {X 0,Y 546.163,Z 370.16,A -85,B 0,C 180,E1 3468.454,E2 3468.454} C_VEL
LIN {X 0,Y 546.113,Z 370.16,A -85,B 0,C 180,E1 3474.395,E2 3474.395} C_VEL
LIN {X 0,Y 546.218,Z 370.16,A -85,B 0,C 180,E1 3480.491,E2 3480.491} C_VEL
LIN {X 0,Y 546.293,Z 370.16,A -85,B 0,C 180,E1 3481.312,E2 3481.312} C_VEL
LIN {X 0,Y 554.065,Z 391.472,A -85,B 0,C 180,E1 3482.077,E2 3482.077} C_VEL
LIN {X 0,Y 553.477,Z 441.88,A -85,B 0,C 180,E1 3482.942,E2 3482.942} C_VEL
LIN {X 0,Y 552.506,Z 478.084,A -85,B 0,C 180,E1 3484.195,E2 3484.195} C_VEL
LIN {X 0,Y 551.175,Z 513.651,A -85,B 0,C 180,E1 3486.097,E2 3486.097} C_VEL
LIN {X 0,Y 549.787,Z 546.441,A -85,B 0,C 180,E1 3488.598,E2 3488.598} C_VEL
LIN {X 0,Y 548.637,Z 574.491,A -85,B 0,C 180,E1 3491.496,E2 3491.496} C_VEL
LIN {X 0,Y 547.749,Z 599.298,A -85,B 0,C 180,E1 3494.946,E2 3494.946} C_VEL
LIN {X 0,Y 547.196,Z 617.475,A -85,B 0,C 180,E1 3498.426,E2 3498.426} C_VEL
LIN {X 0,Y 546.973,Z 630.601,A -85,B 0,C 180,E1 3502.043,E2 3502.043} C_VEL
LIN {X 0,Y 546.868,Z 638.037,A -85,B 0,C 180,E1 3505.283,E2 3505.283} C_VEL
LIN {X 0,Y 546.819,Z 641.508,A -85,B 0,C 180,E1 3508.411,E2 3508.411} C_VEL
LIN {X 0,Y 546.885,Z 641.511,A -85,B 0,C 180,E1 3511.584,E2 3511.584} C_VEL
LIN {X 0,Y 546.874,Z 636.46,A -85,B 0,C 180,E1 3515.558,E2 3515.558} C_VEL
LIN {X 0,Y 547.018,Z 626.846,A -85,B 0,C 180,E1 3519.154,E2 3519.154} C_VEL
LIN {X 0,Y 547.339,Z 611.835,A -85,B 0,C 180,E1 3522.782,E2 3522.782} C_VEL
LIN {X 0,Y 547.931,Z 591.662,A -85,B 0,C 180,E1 3526.243,E2 3526.243} C_VEL
LIN {X 0,Y 548.936,Z 566.074,A -85,B 0,C 180,E1 3529.466,E2 3529.466} C_VEL
LIN {X 0,Y 550.215,Z 536.723,A -85,B 0,C 180,E1 3532.228,E2 3532.228} C_VEL
LIN {X 0,Y 551.651,Z 502.933,A -85,B 0,C 180,E1 3534.553,E2 3534.553} C_VEL
LIN {X 0,Y 552.87,Z 468.202,A -85,B 0,C 180,E1 3536.21,E2 3536.21} C_VEL
LIN {X 0,Y 553.718,Z 432.599,A -85,B 0,C 180,E1 3537.273,E2 3537.273} C_VEL
LIN {X 0,Y 553.3,Z 387.585,A -85,B 0,C 180,E1 3538.021,E2 3538.021} C_VEL
LIN {X 0,Y 546.436,Z 370.16,A -85,B 0,C 180,E1 3538.715,E2 3538.715} C_VEL
LIN {X 0,Y 546.296,Z 370.16,A -85,B 0,C 180,E1 3543.759,E2 3543.759} C_VEL
LIN {X 0,Y 546.159,Z 370.16,A -85,B 0,C 180,E1 3549.606,E2 3549.606} C_VEL
LIN {X 0,Y 546.014,Z 370.16,A -85,B 0,C 180,E1 3556.125,E2 3556.125} C_VEL
LIN {X 0,Y 546.051,Z 370.16,A -85,B 0,C 180,E1 3560.919,E2 3560.919} C_VEL
LIN {X 0,Y 546.101,Z 370.16,A -85,B 0,C 180,E1 3566.327,E2 3566.327} C_VEL
LIN {X 0,Y 546.289,Z 370.16,A -85,B 0,C 180,E1 3572.471,E2 3572.471} C_VEL
LIN {X 0,Y 546.429,Z 370.16,A -85,B 0,C 180,E1 3577.248,E2 3577.248} C_VEL
LIN {X 0,Y 551.183,Z 388.911,A -85,B 0,C 180,E1 3577.736,E2 3577.736} C_VEL
LIN {X 0,Y 550.726,Z 424.138,A -85,B 0,C 180,E1 3578.784,E2 3578.784} C_VEL
LIN {X 0,Y 549.813,Z 456.535,A -85,B 0,C 180,E1 3580.43,E2 3580.43} C_VEL
LIN {X 0,Y 548.789,Z 486.883,A -85,B 0,C 180,E1 3582.748,E2 3582.748} C_VEL
LIN {X 0,Y 547.968,Z 513.018,A -85,B 0,C 180,E1 3585.601,E2 3585.601} C_VEL
LIN {X 0,Y 547.414,Z 532.818,A -85,B 0,C 180,E1 3588.635,E2 3588.635} C_VEL
LIN {X 0,Y 547.075,Z 548.225,A -85,B 0,C 180,E1 3592.046,E2 3592.046} C_VEL
LIN {X 0,Y 546.955,Z 557.122,A -85,B 0,C 180,E1 3595.236,E2 3595.236} C_VEL
LIN {X 0,Y 546.874,Z 561.467,A -85,B 0,C 180,E1 3598.413,E2 3598.413} C_VEL
LIN {X 0,Y 546.835,Z 561.422,A -85,B 0,C 180,E1 3601.585,E2 3601.585} C_VEL
LIN {X 0,Y 546.944,Z 556.773,A -85,B 0,C 180,E1 3604.843,E2 3604.843} C_VEL
LIN {X 0,Y 547.127,Z 546.434,A -85,B 0,C 180,E1 3608.352,E2 3608.352} C_VEL
LIN {X 0,Y 547.462,Z 530.093,A -85,B 0,C 180,E1 3611.767,E2 3611.767} C_VEL
LIN {X 0,Y 548.096,Z 508.85,A -85,B 0,C 180,E1 3614.824,E2 3614.824} C_VEL
LIN {X 0,Y 548.924,Z 483.605,A -85,B 0,C 180,E1 3617.452,E2 3617.452} C_VEL
LIN {X 0,Y 549.907,Z 453.571,A -85,B 0,C 180,E1 3619.668,E2 3619.668} C_VEL
LIN {X 0,Y 550.808,Z 421.12,A -85,B 0,C 180,E1 3621.26,E2 3621.26} C_VEL
LIN {X 0,Y 551.147,Z 386.535,A -85,B 0,C 180,E1 3622.258,E2 3622.258} C_VEL
LIN {X 0,Y 546.301,Z 370.16,A -85,B 0,C 180,E1 3622.754,E2 3622.754} C_VEL
LIN {X 0,Y 546.285,Z 370.16,A -85,B 0,C 180,E1 3628.106,E2 3628.106} C_VEL
LIN {X 0,Y 546.165,Z 370.16,A -85,B 0,C 180,E1 3633.743,E2 3633.743} C_VEL
LIN {X 0,Y 546.251,Z 370.16,A -85,B 0,C 180,E1 3639.599,E2 3639.599} C_VEL
LIN {X 0,Y 546.212,Z 370.16,A -85,B 0,C 180,E1 3646.141,E2 3646.141} C_VEL
LIN {X 0,Y 546.195,Z 370.16,A -85,B 0,C 180,E1 3652.429,E2 3652.429} C_VEL
LIN {X 0,Y 546.158,Z 370.16,A -85,B 0,C 180,E1 3658.222,E2 3658.222} C_VEL
LIN {X 0,Y 546.305,Z 370.16,A -85,B 0,C 180,E1 3663.682,E2 3663.682} C_VEL
LIN {X 0,Y 546.438,Z 370.16,A -85,B 0,C 180,E1 3666.915,E2 3666.915} C_VEL
LIN {X 0,Y 551.891,Z 387.85,A -85,B 0,C 180,E1 3667.523,E2 3667.523} C_VEL
LIN {X 0,Y 551.308,Z 421.177,A -85,B 0,C 180,E1 3668.522,E2 3668.522} C_VEL
LIN {X 0,Y 550.205,Z 452.755,A -85,B 0,C 180,E1 3670.118,E2 3670.118} C_VEL
LIN {X 0,Y 549.055,Z 480.764,A -85,B 0,C 180,E1 3672.19,E2 3672.19} C_VEL
LIN {X 0,Y 548.107,Z 507.507,A -85,B 0,C 180,E1 3674.913,E2 3674.913} C_VEL
LIN {X 0,Y 547.473,Z 528.239,A -85,B 0,C 180,E1 3677.83,E2 3677.83} C_VEL
LIN {X 0,Y 547.121,Z 543.56,A -85,B 0,C 180,E1 3680.847,E2 3680.847} C_VEL
LIN {X 0,Y 546.928,Z 554.503,A -85,B 0,C 180,E1 3684.084,E2 3684.084} C_VEL
LIN {X 0,Y 546.842,Z 559.886,A -85,B 0,C 180,E1 3686.828,E2 3686.828} C_VEL
LIN {X 0,Y 546.879,Z 561.997,A -85,B 0,C 180,E1 3690.002,E2 3690.002} C_VEL
LIN {X 0,Y 546.862,Z 559.743,A -85,B 0,C 180,E1 3693.176,E2 3693.176} C_VEL
LIN {X 0,Y 546.987,Z 553.029,A -85,B 0,C 180,E1 3696.359,E2 3696.359} C_VEL
LIN {X 0,Y 547.138,Z 541.416,A -85,B 0,C 180,E1 3699.559,E2 3699.559} C_VEL
LIN {X 0,Y 547.568,Z 523.855,A -85,B 0,C 180,E1 3702.781,E2 3702.781} C_VEL
LIN {X 0,Y 548.323,Z 501.575,A -85,B 0,C 180,E1 3705.681,E2 3705.681} C_VEL
LIN {X 0,Y 549.465,Z 472.145,A -85,B 0,C 180,E1 3708.434,E2 3708.434} C_VEL
LIN {X 0,Y 550.639,Z 442.066,A -85,B 0,C 180,E1 3710.41,E2 3710.41} C_VEL
LIN {X 0,Y 551.659,Z 410.707,A -85,B 0,C 180,E1 3711.764,E2 3711.764} C_VEL
LIN {X 0,Y 550.992,Z 384.079,A -85,B 0,C 180,E1 3712.512,E2 3712.512} C_VEL
LIN {X 0,Y 546.347,Z 370.16,A -85,B 0,C 180,E1 3713.023,E2 3713.023} C_VEL
LIN {X 0,Y 546.216,Z 370.16,A -85,B 0,C 180,E1 3718.114,E2 3718.114} C_VEL
LIN {X 0,Y 546.145,Z 370.16,A -85,B 0,C 180,E1 3723.739,E2 3723.739} C_VEL
LIN {X 0,Y 546.063,Z 370.16,A -85,B 0,C 180,E1 3729.621,E2 3729.621} C_VEL
LIN {X 0,Y 546.171,Z 370.16,A -85,B 0,C 180,E1 3736.136,E2 3736.136} C_VEL
LIN {X 0,Y 546.132,Z 370.16,A -85,B 0,C 180,E1 3742.423,E2 3742.423} C_VEL
LIN {X 0,Y 546.114,Z 370.16,A -85,B 0,C 180,E1 3748.218,E2 3748.218} C_VEL
LIN {X 0,Y 546.304,Z 370.16,A -85,B 0,C 180,E1 3753.681,E2 3753.681} C_VEL
LIN {X 0,Y 546.4,Z 370.16,A -85,B 0,C 180,E1 3758.889,E2 3758.889} C_VEL
LIN {X 0,Y 546.475,Z 370.16,A -85,B 0,C 180,E1 3763.918,E2 3763.918} C_VEL
LIN {X 0,Y 546.444,Z 370.16,A -85,B 0,C 180,E1 3768.819,E2 3768.819} C_VEL
LIN {X 0,Y 546.474,Z 370.16,A -85,B 0,C 180,E1 3773.639,E2 3773.639} C_VEL
LIN {X 0,Y 546.507,Z 370.16,A -85,B 0,C 180,E1 3778.414,E2 3778.414} C_VEL
LIN {X 0,Y 546.495,Z 370.16,A -85,B 0,C 180,E1 3783.177,E2 3783.177} C_VEL
LIN {X 0,Y 546.423,Z 370.16,A -85,B 0,C 180,E1 3787.964,E2 3787.964} C_VEL
LIN {X 0,Y 546.382,Z 370.16,A -85,B 0,C 180,E1 3792.808,E2 3792.808} C_VEL
LIN {X 0,Y 546.301,Z 370.16,A -85,B 0,C 180,E1 3797.983,E2 3797.983} C_VEL
LIN {X 0,Y 546.32,Z 370.16,A -85,B 0,C 180,E1 3801.548,E2 3801.548} C_VEL
LIN {X 0,Y 542.323,Z 370.16,A -85,B 0,C 180,E1 3803.337,E2 3803.337} C_VEL
LIN {X 0,Y 538.361,Z 370.16,A -85,B 0,C 180,E1 3805.152,E2 3805.152} C_VEL
LIN {X 0,Y 538.23,Z 370.16,A -85,B 0,C 180,E1 3810.419,E2 3810.419} C_VEL
LIN {X 0,Y 538.304,Z 370.16,A -85,B 0,C 180,E1 3816.201,E2 3816.201} C_VEL
LIN {X 0,Y 538.144,Z 370.16,A -85,B 0,C 180,E1 3822.469,E2 3822.469} C_VEL
LIN {X 0,Y 538.183,Z 370.16,A -85,B 0,C 180,E1 3827.533,E2 3827.533} C_VEL
LIN {X 0,Y 538.218,Z 370.16,A -85,B 0,C 180,E1 3833.79,E2 3833.79} C_VEL
LIN {X 0,Y 538.235,Z 370.16,A -85,B 0,C 180,E1 3839.58,E2 3839.58} C_VEL
LIN {X 0,Y 538.394,Z 370.832,A -85,B 0,C 180,E1 3840.881,E2 3840.881} C_VEL
LIN {X 0,Y 546.948,Z 391.965,A -85,B 0,C 180,E1 3841.688,E2 3841.688} C_VEL
LIN {X 0,Y 546.437,Z 441.231,A -85,B 0,C 180,E1 3842.546,E2 3842.546} C_VEL
LIN {X 0,Y 545.345,Z 477.159,A -85,B 0,C 180,E1 3843.788,E2 3843.788} C_VEL
LIN {X 0,Y 543.917,Z 511.973,A -85,B 0,C 180,E1 3845.649,E2 3845.649} C_VEL
LIN {X 0,Y 542.379,Z 545.288,A -85,B 0,C 180,E1 3848.184,E2 3848.184} C_VEL
LIN {X 0,Y 541.082,Z 572.738,A -85,B 0,C 180,E1 3851.016,E2 3851.016} C_VEL
LIN {X 0,Y 540.058,Z 596.961,A -85,B 0,C 180,E1 3854.344,E2 3854.344} C_VEL
LIN {X 0,Y 539.428,Z 615.713,A -85,B 0,C 180,E1 3857.846,E2 3857.846} C_VEL
LIN {X 0,Y 539.155,Z 629.454,A -85,B 0,C 180,E1 3861.52,E2 3861.52} C_VEL
LIN {X 0,Y 538.978,Z 637.962,A -85,B 0,C 180,E1 3865.164,E2 3865.164} C_VEL
LIN {X 0,Y 538.933,Z 641.508,A -85,B 0,C 180,E1 3868.388,E2 3868.388} C_VEL
LIN {X 0,Y 538.994,Z 641.511,A -85,B 0,C 180,E1 3871.607,E2 3871.607} C_VEL
LIN {X 0,Y 538.998,Z 637.971,A -85,B 0,C 180,E1 3874.831,E2 3874.831} C_VEL
LIN {X 0,Y 539.148,Z 628.183,A -85,B 0,C 180,E1 3878.882,E2 3878.882} C_VEL
LIN {X 0,Y 539.457,Z 613.792,A -85,B 0,C 180,E1 3882.56,E2 3882.56} C_VEL
LIN {X 0,Y 540.103,Z 594.34,A -85,B 0,C 180,E1 3886.067,E2 3886.067} C_VEL
LIN {X 0,Y 541.223,Z 569.267,A -85,B 0,C 180,E1 3889.398,E2 3889.398} C_VEL
LIN {X 0,Y 542.612,Z 539.248,A -85,B 0,C 180,E1 3892.34,E2 3892.34} C_VEL
LIN {X 0,Y 544.205,Z 506.948,A -85,B 0,C 180,E1 3894.661,E2 3894.661} C_VEL
LIN {X 0,Y 545.622,Z 470.964,A -85,B 0,C 180,E1 3896.475,E2 3896.475} C_VEL
LIN {X 0,Y 546.665,Z 433.772,A -85,B 0,C 180,E1 3897.628,E2 3897.628} C_VEL
LIN {X 0,Y 546.462,Z 390.023,A -85,B 0,C 180,E1 3898.368,E2 3898.368} C_VEL
LIN {X 0,Y 538.452,Z 370.16,A -85,B 0,C 180,E1 3899.192,E2 3899.192} C_VEL
LIN {X 0,Y 538.33,Z 370.16,A -85,B 0,C 180,E1 3905.357,E2 3905.357} C_VEL
LIN {X 0,Y 538.156,Z 370.16,A -85,B 0,C 180,E1 3910.574,E2 3910.574} C_VEL
LIN {X 0,Y 538.046,Z 370.16,A -85,B 0,C 180,E1 3917.015,E2 3917.015} C_VEL
LIN {X 0,Y 538.153,Z 370.16,A -85,B 0,C 180,E1 3921.967,E2 3921.967} C_VEL
LIN {X 0,Y 538.19,Z 370.16,A -85,B 0,C 180,E1 3927.691,E2 3927.691} C_VEL
LIN {X 0,Y 538.387,Z 370.16,A -85,B 0,C 180,E1 3933.261,E2 3933.261} C_VEL
LIN {X 0,Y 538.511,Z 370.16,A -85,B 0,C 180,E1 3936.981,E2 3936.981} C_VEL
LIN {X 0,Y 543.694,Z 390.392,A -85,B 0,C 180,E1 3937.509,E2 3937.509} C_VEL
LIN {X 0,Y 543.191,Z 424.769,A -85,B 0,C 180,E1 3938.547,E2 3938.547} C_VEL
LIN {X 0,Y 542.278,Z 456.695,A -85,B 0,C 180,E1 3940.181,E2 3940.181} C_VEL
LIN {X 0,Y 541.218,Z 485.804,A -85,B 0,C 180,E1 3942.394,E2 3942.394} C_VEL
LIN {X 0,Y 540.283,Z 509.877,A -85,B 0,C 180,E1 3944.987,E2 3944.987} C_VEL
LIN {X 0,Y 539.624,Z 530.609,A -85,B 0,C 180,E1 3948.058,E2 3948.058} C_VEL
LIN {X 0,Y 539.265,Z 546.745,A -85,B 0,C 180,E1 3951.523,E2 3951.523} C_VEL
LIN {X 0,Y 539.093,Z 557.113,A -85,B 0,C 180,E1 3955.166,E2 3955.166} C_VEL
LIN {X 0,Y 538.983,Z 561.459,A -85,B 0,C 180,E1 3958.389,E2 3958.389} C_VEL
LIN {X 0,Y 538.946,Z 561.422,A -85,B 0,C 180,E1 3961.609,E2 3961.609} C_VEL
LIN {X 0,Y 539.069,Z 556.939,A -85,B 0,C 180,E1 3964.832,E2 3964.832} C_VEL
LIN {X 0,Y 539.27,Z 546.44,A -85,B 0,C 180,E1 3968.474,E2 3968.474} C_VEL
LIN {X 0,Y 539.619,Z 530.088,A -85,B 0,C 180,E1 3971.94,E2 3971.94} C_VEL
LIN {X 0,Y 540.368,Z 508.898,A -85,B 0,C 180,E1 3975.041,E2 3975.041} C_VEL
LIN {X 0,Y 541.302,Z 483.687,A -85,B 0,C 180,E1 3977.706,E2 3977.706} C_VEL
LIN {X 0,Y 542.348,Z 454.147,A -85,B 0,C 180,E1 3979.903,E2 3979.903} C_VEL
LIN {X 0,Y 543.359,Z 421.093,A -85,B 0,C 180,E1 3981.54,E2 3981.54} C_VEL
LIN {X 0,Y 543.406,Z 387.012,A -85,B 0,C 180,E1 3982.545,E2 3982.545} C_VEL
LIN {X 0,Y 538.393,Z 370.16,A -85,B 0,C 180,E1 3983.098,E2 3983.098} C_VEL
LIN {X 0,Y 538.313,Z 370.16,A -85,B 0,C 180,E1 3988.56,E2 3988.56} C_VEL
LIN {X 0,Y 538.24,Z 370.16,A -85,B 0,C 180,E1 3994.23,E2 3994.23} C_VEL
LIN {X 0,Y 538.376,Z 370.16,A -85,B 0,C 180,E1 3998.215,E2 3998.215} C_VEL
LIN {X 0,Y 538.197,Z 370.16,A -85,B 0,C 180,E1 4004.685,E2 4004.685} C_VEL
LIN {X 0,Y 538.212,Z 370.16,A -85,B 0,C 180,E1 4009.69,E2 4009.69} C_VEL
LIN {X 0,Y 538.178,Z 370.16,A -85,B 0,C 180,E1 4015.766,E2 4015.766} C_VEL
LIN {X 0,Y 538.297,Z 370.16,A -85,B 0,C 180,E1 4021.44,E2 4021.44} C_VEL
LIN {X 0,Y 538.502,Z 370.16,A -85,B 0,C 180,E1 4026.478,E2 4026.478} C_VEL
LIN {X 0,Y 544.871,Z 390.162,A -85,B 0,C 180,E1 4027.188,E2 4027.188} C_VEL
LIN {X 0,Y 544.184,Z 423.877,A -85,B 0,C 180,E1 4028.249,E2 4028.249} C_VEL
LIN {X 0,Y 542.902,Z 454.772,A -85,B 0,C 180,E1 4029.87,E2 4029.87} C_VEL
